// TIA Portal project "CmDrvSerPosRev0.0.5" (V15.1)

(* hardware
DEVICE "S7-1200 station_1"  S7-1200 Station
   slot 0: "Rack_0"  S7-1200 Rack  Rack  V1.0
   slot 1: "CPU"  CPU 1215C DC/DC/DC  6ES7 215-1AG40-0XB0  V4.2
DEVICE "GSD-Geraet_6"  GSD.Device.PN
   slot 0: "Baugruppenträger"  Rail  V1.0
   slot 0: "rlp_drv_ser_nip_rev1_id180303002"  E84AYCER  V 2.1
DEVICE "HMI"  TP700 Comfort
   slot 0: "HMI"  TP700 Comfort  6AV2 124-0GC01-0AX0  15.1.0.0
   slot 1: "HMI_RT_1"  TP700 Comfort  6AV2 124-0GC01-0AX0  15.1.0.0
   slot 5: "HMI.IE_CP_1"  PROFINET Interface  15.0.1.0
      slot 1: "PROFINET Interface_1"  PROFINET Interface
         slot 1: "Port_1"  Port
         slot 2: "Port_2"  Port
   slot 7: "HMI.MPI/DP_CP_1"  MPI/DP Interface  15.0.1.0
*)

// ===== PLC "CPU"  CPU 1215C DC/DC/DC =====

VAR_GLOBAL   // PLC tag table "Default tag table"
   "di_PbStart" AT %I0.0 : Bool;
   "di_PbStop" AT %I0.1 : Bool;
   "di_PbReset" AT %I0.2 : Bool;
   "di_PbJog" AT %I0.3 : Bool;
   "di_FeedbackEmStop" AT %I0.4 : Bool;   // 1 = EmStop / 0 = EmStopOK
   "dq_EnableDrive" AT %Q0.5 : Bool;
END_VAR

TYPE "stcCmDrvSerPos_CD"
   STRUCT
      iModeSet : Int;
      iStartAreaAdressErrorID : Int;   // Range between 0..64
      Commands : "stcCmCommand";
      Recipe : "stcCmDrvSerPos_RECIPE";
   END_STRUCT;
END_TYPE

TYPE "stcCmCommon_VIS"
VERSION : 0.1
   STRUCT
      stc_NewTimeToSet : Struct
         year : UInt;
         month : USInt;
         day : USInt;
         weekday : USInt;
         hour : USInt;
         minute : USInt;
         iq_bRequestLoadNewTime : Bool;
      END_STRUCT;
      q_dtlActualPlcSystemTime : DTL;
      q_rActualPlcCycleTime_Sec : Real;
   END_STRUCT;
END_TYPE

TYPE "stcCmCommon_SW"
VERSION : 0.1
   STRUCT
      q_dtlActualPlcSystem_Time : DTL;
      q_rActualPlcCycleTime_Sec : Real;
      q_bSyncBlink : Bool;   // Signal light Indicator blink
      q_bSyncBlinkText : Bool;   // Hmi status text scroll, swap, refresh blink
      q_bSyncPulsText : Bool;   // Puls is true for one cpu cycle
      q_bAlwaysTrue : Bool := TRUE;
      q_bAlwaysFalse : Bool := FALSE;
   END_STRUCT;
END_TYPE

TYPE "stcCmDrvSerPos_VIS"
   STRUCT
      Commands : "stcCmCommand";
      Interlocks : "stcCmCommand";
      Indicators : "stcCmIndicators";
      Recipe : "stcCmDrvSerPos_RECIPE";
      Settings : "stcCmDrvSerPos_CFG";
      CD : "stcCmDrvSerPos_CD";
      SD : "stcCmDrvSerPos_SD";
      bLimitsSwitchPositiveActivated : Bool;   // Module specific
      bLimitsSwitchNegativeActivated : Bool;   // Module specific
      bHomingSensorActivated : Bool;   // Module specific
   END_STRUCT;
END_TYPE

TYPE "stcCmDrvSerPos_RETAIN"
   STRUCT
      Recipe : "stcCmDrvSerPos_RECIPE";
      Settings : "stcCmDrvSerPos_CFG";
      ErrorWarningReleased : Bool;
   END_STRUCT;
END_TYPE

TYPE "stcCmDrvSerPos_RECIPE"
   STRUCT
      rSpPosition_Units : Real;
   END_STRUCT;
END_TYPE

TYPE "stcCmDrvSerPos_CFG"
   STRUCT
      rSpLimitH_Units : Real;
      rSpLimitL_Units : Real;
      rSpPositionOffset_Units : Real;
      iSetUnits : Int;   // 0=um, 1=mm, 2=cm, 10=mil, 11=Inch, 12=foot
   END_STRUCT;
END_TYPE

TYPE "stcCmDrvSerPos_SD"
   STRUCT
      iModeActual : Int;
      iModuleState : Int;
      bRFR : Bool;   // Ready for run AND active mode is Automatic
      bExecuting : Bool;   // PosCtrl executing = Executing production AND , active mode is Automatic
      bRecipeAccepted : Bool;   // Recipe as setpoints are accepted and equal with active internal setpoints
      ErrorWarningReleased : Bool;   // ErrorWarning enabled
      CommandsActivated : "stcCmCommand";   // Feedback of commands while there are activated in the StateCases
      Recipe : "stcCmDrvSerPos_RECIPE";
      ProcessValue : "stcCmDrvSerPos_PROCESS";
      ErrorWarning : "stcCmErrorWarning";
   END_STRUCT;
END_TYPE

TYPE "stcCmDrvSerPos_REMOTE"
   STRUCT
      ErrorID : DInt;
      iModuleState : Int;
      Recipe : "stcCmDrvSerPos_RECIPE";
      Process : "stcCmDrvSerPos_PROCESS";
   END_STRUCT;
END_TYPE

TYPE "stcCmDrvSerPos_PROCESS"
   STRUCT
      rPvPosition_Units : Real;
   END_STRUCT;
END_TYPE

// folder: OEM

TYPE "stcLCB_12x_SetAxisData_Sw"
VERSION : 0.1
   STRUCT
      rUnitsToPos : Real;
      rPosToUnits : Real;
   END_STRUCT;
END_TYPE

// folder: Template_ControlModule

TYPE "stcCmStates"
   STRUCT
      iModule : Int;
      iInit : Int;   // Initializing/PowerUp
      iReady : Int;
      iEnableDisable : Int;
      iJogFwdCwUpLoading : Int;
      iJogRevCcwDownUnloading : Int;
      iHoming : Int;
      iExecutingAutomatic : Int;   // Position control active, Conveyor is executing, Cutter is executing
      iError : Int;
   END_STRUCT;
END_TYPE

TYPE "stcCmCommand"
   STRUCT
      ModeChange : Bool;
      Enable : Bool;
      Disable : Bool;
      JogFwdCwUpLoading : Bool;
      JogRevCcwDownUnloading : Bool;
      StartHoming : Bool;
      StopHoming : Bool;
      StartExecuteAutomatic : Bool;   // Position control active, Conveyor is executing, Cutter is executing
      StopExecuteAutomatic : Bool;   // Position control active, Conveyor is executing, Cutter is executing
      EnableReleaseErrorWarning : Bool;
      DisableReleaseErrorWarning : Bool;
      ExecuteLoadRecipe : Bool;   // Execute module to recipe value
      ManualToAutomatic : Bool;   // Set module from Temporarily Manual control into automatic so it is reacting at commands from heigher layer
      AutomaticToManual : Bool;   // Temporarily Set module from Automatic into Manual control. The module react at VIS commands and not from heigher layer commands
      PbReset : Bool;
      PbSingleStep : Bool;   // At falling edge of the push button, the single step command will react in mode=5=SingleStepMode
   END_STRUCT;
END_TYPE

TYPE "stcCmIndicators"
   STRUCT
      PushButtons : "stcCmCommand";
      Status : Struct
         IsEnabled : Bool;
         IsHomed : Bool;
         BusyJogFwdCwUpLoading : Bool;
         BusyJogRevCcwDownUnloading : Bool;
         IsAtTargetPosSpeed : Bool;
      END_STRUCT;
   END_STRUCT;
END_TYPE

TYPE "stcCmErrorWarning"
   STRUCT
      diModuleErrorID : DInt;   // bit0-15=ErrorID, bit16-25ErrorSubjectArea, bit26-31 location area
      bErrorTripped : Bool;   // There is one or more error's going on
      bWarningTripped : Bool;   // There is one or more warning's going on
      wError : Word;   // 16 bit word. Each idividual bit stands for a item
      wWarning : Word;   // 16 bit word. Each idividual bit stands for a item
      iAdressAreaSize : Int;   // Range 0..64. the count of error location areas inside the module
   END_STRUCT;
END_TYPE

// folder: (top level)

DATA_BLOCK "DB_CmCommon"   // DB1
{ S7_Optimized_Access := 'TRUE' }
VERSION : 0.1
// stored: InstanceOfName CmCommon
"CmCommon"
BEGIN
END_DATA_BLOCK

DATA_BLOCK "DB_CmDrvSerPos"   // DB2
{ S7_Optimized_Access := 'TRUE' }
VERSION : 0.1
// stored: InstanceOfName CmDrvSerPos
"CmDrvSerPos"
BEGIN
END_DATA_BLOCK

DATA_BLOCK "VIS_CmDrvSerPos"   // DB3
{ S7_Optimized_Access := 'TRUE' }
VERSION : 0.1
   VAR
      stc : "stcCmDrvSerPos_VIS";
   END_VAR
BEGIN
END_DATA_BLOCK

DATA_BLOCK "VIS_CmCommon"   // DB4
{ S7_Optimized_Access := 'TRUE' }
VERSION : 0.1
   VAR
      stc : "stcCmCommon_VIS";
   END_VAR
BEGIN
END_DATA_BLOCK

DATA_BLOCK "RETAIN_CmDrvSerPos"   // DB5
{ S7_Optimized_Access := 'TRUE' }
VERSION : 0.1
   VAR RETAIN
      stc : "stcCmDrvSerPos_RETAIN";
   END_VAR
BEGIN
   stc.Recipe.rSpPosition_Units := 150.0;
   stc.Settings.rSpLimitH_Units := 300.0;
   stc.Settings.rSpLimitL_Units := 4.0;
   stc.Settings.rSpPositionOffset_Units := -1.8;
   stc.Settings.iSetUnits := 0;
END_DATA_BLOCK

FUNCTION_BLOCK "CmDrvSerPos"   // FB1, FBD
TITLE = Control Module: Drive Servo Positioning OEM: LENZE
{ S7_Optimized_Access := 'TRUE' }
VERSION : 0.1
   VAR_INPUT
      i_HW_IO_Head : Hw_Io;
      i_bPbReset : Bool;
      i_bQuickStop : Bool;   // True is quickstop situation active, False is normal operating
      i_bPbSingleStep : Bool;   // At falling edge of the push button, the single step command will react in mode=5=SingleStepMode
      i_JogFwdCwUpLoading : Bool;
      i_JogRevCcwDownUnloading : Bool;
      Common : "stcCmCommon_SW";
      CD : "stcCmDrvSerPos_CD";
   END_VAR
   VAR_OUTPUT
      SD : "stcCmDrvSerPos_SD";
      q_bDriveIEnableRfr : Bool;   // True=Drive from InhibitSleepMode into RFR, False=Inhibit Sleep situation en drive stopped functioning
   END_VAR
   VAR_IN_OUT
      VIS : "stcCmDrvSerPos_VIS";
      RETAIN : "stcCmDrvSerPos_RETAIN";
   END_VAR
   VAR
      RM : "stcCmDrvSerPos_CD";
      FM : Struct
         Interlock : "stcCmCommand";
         ModeActual : Int;
      END_STRUCT;
      FS : Struct
         StateCases : "stcCmStates";
         StateCasesPrevious : "stcCmStates";
         Commands : "stcCmCommand";
         CommandsActive : "stcCmCommand";
         Indicators : "stcCmIndicators";
         Settings : "stcCmDrvSerPos_CFG";
         Recipe : "stcCmDrvSerPos_RECIPE";
         ProcessValues : "stcCmDrvSerPos_PROCESS";
         ErrorWarningModule : "stcCmErrorWarning";
         ErrorWarning : "stcCmErrorWarning";
         Intern : Struct
            rPreviousSpPosition_Units : Real;
            ErrorWarningReleased : Bool;
            ErrorWarning : Struct
               wErrorLocationArea : Word;
               wErrorSubjectArea : Word;
               wErrorID : Word;
               dwModuleErrorID : DWord;
               bErrorTripped : Bool;
               bWarningTripped : Bool;
            END_STRUCT;
         END_STRUCT;
         Outputs : Struct
            bDriveInhibitTerminal : Bool;   // True=Drive from InhibitSleepMode into RFR, False=Inhibit Sleep situation en drive stopped functioning
         END_STRUCT;
      END_STRUCT;
      InstanceOEM_LCB_12x_SetAxisData : "LCB_12x_SetAxisData";
      InstanceOEM_LCB_12x_TablePositioning_V2 : "LCB_12x_TablePositioning_V2";
      InstanceF_TRIG_PbSingleStep : F_TRIG;
      InstanceR_TRIG_cmdEnable : R_TRIG;
      InstanceR_TRIG_cmdDisable : R_TRIG;
      InstanceR_TRIG_cmdStartHoming : R_TRIG;
      InstanceR_TRIG_cmdStopHoming : R_TRIG;
      InstanceR_TRIG_cmdStartExecAutomatic : R_TRIG;
      InstanceR_TRIG_cmdStopExecAutomatic : R_TRIG;
      InstanceR_TRIG_cmdLoadRecipe : R_TRIG;
   END_VAR
BEGIN

REGION Network 1 (SCL): Resource Manager
   // Mapping data channels --> Data channel switch depending of actual Mode
   CASE #FM.ModeActual OF

       0: //Wrong Mode
           #RM.iModeSet := #CD.iModeSet;
           //
           #RM.Commands.ModeChange := #CD.Commands.ModeChange;
           #RM.Commands.Enable :=
           #RM.Commands.Disable :=
           #RM.Commands.JogFwdCwUpLoading :=
           #RM.Commands.JogRevCcwDownUnloading :=
           #RM.Commands.StartHoming :=
           #RM.Commands.StopHoming :=
           #RM.Commands.StartExecuteAutomatic :=
           #RM.Commands.StopExecuteAutomatic :=
           #RM.Commands.EnableReleaseErrorWarning :=
           #RM.Commands.DisableReleaseErrorWarning :=
           #RM.Commands.ExecuteLoadRecipe :=
           #RM.Commands.ManualToAutomatic :=
           #RM.Commands.AutomaticToManual := FALSE;
           #RM.Commands.PbReset :=
               #CD.Commands.PbReset OR
               #VIS.Commands.PbReset OR
               #i_bPbReset;
           #RM.Commands.PbSingleStep := FALSE;

       1: //Automatic Inline
           #RM.iModeSet := #CD.iModeSet;
           #RM.Commands := #CD.Commands;
           //Overrule single commands
           #RM.Commands.PbReset :=
               #CD.Commands.PbReset OR
               #VIS.Commands.PbReset OR
               #i_bPbReset;

       2: //Automatic standalone
           #RM.iModeSet := #CD.iModeSet;
           #RM.Commands := #CD.Commands;
           //Overrule single commands
           #RM.Commands.PbReset :=
               #CD.Commands.PbReset OR
               #VIS.Commands.PbReset OR
               #i_bPbReset;

       3: //Manual
           #RM.iModeSet := #CD.iModeSet;
           #RM.Commands := #VIS.Commands;
           #RM.Commands.ModeChange := #CD.Commands.ModeChange;
           //Overrule single commands
           #RM.Commands.PbReset :=
               #CD.Commands.PbReset OR
               #VIS.Commands.PbReset OR
               #i_bPbReset;
           #RM.Commands.JogFwdCwUpLoading :=
               #VIS.Commands.JogFwdCwUpLoading OR
               #CD.Commands.JogFwdCwUpLoading OR
               #i_JogFwdCwUpLoading;
           #RM.Commands.JogRevCcwDownUnloading :=
               #VIS.Commands.JogRevCcwDownUnloading OR
               #CD.Commands.JogRevCcwDownUnloading OR
               #i_JogRevCcwDownUnloading;

       4: //Service
           #RM.iModeSet := #CD.iModeSet;
           #RM.Commands := #VIS.Commands;
           #RM.Commands.ModeChange := #CD.Commands.ModeChange;
           //Overrule single commands
           #RM.Commands.PbReset :=
               #CD.Commands.PbReset OR
               #VIS.Commands.PbReset OR
               #i_bPbReset;
           #RM.Commands.JogFwdCwUpLoading :=
               #VIS.Commands.JogFwdCwUpLoading OR
               #CD.Commands.JogFwdCwUpLoading OR
               #i_JogFwdCwUpLoading;
           #RM.Commands.JogRevCcwDownUnloading :=
               #VIS.Commands.JogRevCcwDownUnloading OR
               #CD.Commands.JogRevCcwDownUnloading OR
               #i_JogRevCcwDownUnloading;

       5: //SingleStep
           #RM.iModeSet := #CD.iModeSet;
           #RM.Commands := #VIS.Commands;
           #RM.Commands.ModeChange := #CD.Commands.ModeChange;
           //Overrule single commands
           #RM.Commands.PbReset :=
               #CD.Commands.PbReset OR
               #VIS.Commands.PbReset OR
               #i_bPbReset;
           #RM.Commands.JogFwdCwUpLoading :=
               #VIS.Commands.JogFwdCwUpLoading OR
               #CD.Commands.JogFwdCwUpLoading OR
               #i_JogFwdCwUpLoading;
           #RM.Commands.JogRevCcwDownUnloading :=
               #VIS.Commands.JogRevCcwDownUnloading OR
               #CD.Commands.JogRevCcwDownUnloading OR
               #i_JogRevCcwDownUnloading;
           #RM.Commands.PbReset :=
               #CD.Commands.PbReset OR
               #VIS.Commands.PbReset OR
               #i_bPbReset;
           #RM.Commands.PbSingleStep :=
               #CD.Commands.PbSingleStep OR
               #VIS.Commands.PbSingleStep OR
               #i_bPbSingleStep;
   END_CASE;
END_REGION

REGION Network 2 (SCL): Funtional Manager: Interlocks
   REGION #FM.Interlock.ModeChange
       #FM.Interlock.ModeChange :=
           (
           #FS.StateCases.iModule = 10 (*Disabled*)OR
           #FS.StateCases.iModule = 30 (*ReadyEnabled*) OR
           #FS.StateCases.iModule = 70 (*ReadyHomed*) OR
           #FS.StateCases.iModule = 80 (*Executing*) 
           );
   END_REGION

   REGION #FM.Interlock.Enable Disable
       #FM.Interlock.Disable :=
           (
           #FS.StateCases.iInit = 100 AND
           #FS.StateCases.iReady > 0 AND
           #FS.StateCases.iEnableDisable > 0 AND
           #FS.StateCases.iJogFwdCwUpLoading = 0 AND
           #FS.StateCases.iJogRevCcwDownUnloading = 0 AND
           (#FS.StateCases.iHoming = 0 OR #FS.StateCases.iHoming = 100) AND
           #FS.StateCases.iExecutingAutomatic = 0
           );

       #FM.Interlock.Enable :=
           (
           #FS.StateCases.iInit = 100 AND
           #FS.StateCases.iReady > 0 AND
           #FS.StateCases.iEnableDisable = 0 AND
           #FS.StateCases.iJogFwdCwUpLoading = 0 AND
           #FS.StateCases.iJogRevCcwDownUnloading = 0 AND
           (#FS.StateCases.iHoming = 0 OR #FS.StateCases.iHoming = 100) AND
           #FS.StateCases.iExecutingAutomatic = 0
           );
   END_REGION

   REGION #FM.Interlock.Jog
       #FM.Interlock.JogFwdCwUpLoading :=
       (
       #FM.ModeActual <> 5 (*Single step mode*)AND
       #FS.StateCases.iInit = 100 AND
       #FS.StateCases.iReady >= 20 AND
       #FS.StateCases.iEnableDisable = 100(*Executed*)AND
       // #FS.State.iJogFwdCwUp = 0 AND
       #FS.StateCases.iJogRevCcwDownUnloading = 0 AND
       (#FS.StateCases.iHoming = 0 OR #FS.StateCases.iHoming = 100 (*Executed*)) AND
       #FS.StateCases.iExecutingAutomatic = 0 AND
       (#FS.StateCases.iError = 0 (*No Error*) OR #FS.StateCases.iError >= 500) (*Warning*) AND
       NOT #InstanceOEM_LCB_12x_TablePositioning_V2.xHW_LimitSwitchPos
       );

       #FM.Interlock.JogRevCcwDownUnloading :=
       (
       #FM.ModeActual <> 5 (*Single step mode*)AND
       #FS.StateCases.iInit = 100 AND
       #FS.StateCases.iReady >= 20 AND
       #FS.StateCases.iEnableDisable = 100(*Executed*)AND
       #FS.StateCases.iJogFwdCwUpLoading = 0 AND
       //#FS.State.iJogRevCcwDown = 0 AND
       (#FS.StateCases.iHoming = 0 OR #FS.StateCases.iHoming = 100 (*Executed*)) AND
       #FS.StateCases.iExecutingAutomatic = 0 AND
       (#FS.StateCases.iError = 0 (*No Error*) OR #FS.StateCases.iError >= 500) (*Warning*) AND
       NOT #InstanceOEM_LCB_12x_TablePositioning_V2.xHW_LimitSwitchNeg
       );
   END_REGION

   REGION #FM.Interlock.Homing Start Stop
       #FM.Interlock.StartHoming :=
           (
           #FS.StateCases.iInit = 100 AND
           #FS.StateCases.iReady >= 20 AND
           #FS.StateCases.iEnableDisable = 100(*Executed*)AND
           #FS.StateCases.iJogFwdCwUpLoading = 0 AND
           #FS.StateCases.iJogRevCcwDownUnloading = 0 AND
           (#FS.StateCases.iHoming = 0 OR #FS.StateCases.iHoming = 100 (*Executed*)) AND
           #FS.StateCases.iExecutingAutomatic = 0 AND
           #FS.StateCases.iError = 0
           );

       #FM.Interlock.StopHoming :=
           (
           #FS.StateCases.iInit = 100 AND
           #FS.StateCases.iReady >= 20 AND
           #FS.StateCases.iEnableDisable = 100(*Executed*)AND
           #FS.StateCases.iJogFwdCwUpLoading = 0 AND
           #FS.StateCases.iJogRevCcwDownUnloading = 0 AND
           #FS.StateCases.iHoming > 0 (*Stopped*) AND
           #FS.StateCases.iExecutingAutomatic = 0 AND
           #FS.StateCases.iError = 0
           );
   END_REGION

   REGION #FM.Interlock.PositionControl Start Stop
       #FM.Interlock.StartExecuteAutomatic :=
           (
           #FS.StateCases.iInit = 100 AND
           #FS.StateCases.iReady >= 30 AND
           #FS.StateCases.iEnableDisable = 100(*Executed*)AND
           #FS.StateCases.iJogFwdCwUpLoading = 0 AND
           #FS.StateCases.iJogRevCcwDownUnloading = 0 AND
           #FS.StateCases.iHoming = 100 (*Executed*) AND
           #FS.StateCases.iExecutingAutomatic = 0 (*Stopped*)AND
           #FS.StateCases.iError = 0
           );

       #FM.Interlock.StopExecuteAutomatic :=
           (
           #FS.StateCases.iInit = 100 AND
           //#FS.State.iReady > 0 AND
           #FS.StateCases.iEnableDisable = 100(*Executed*)AND
           #FS.StateCases.iJogFwdCwUpLoading = 0 AND
           #FS.StateCases.iJogRevCcwDownUnloading = 0 AND
           #FS.StateCases.iHoming = 100 (*Executed*)AND
           #FS.StateCases.iExecutingAutomatic > 0 (*Stopped*) AND
           #FS.StateCases.iError = 0
           );
   END_REGION

   REGION #FM.Interlock.ReleaseErrorWarning
       #FM.Interlock.EnableReleaseErrorWarning :=
           (
           #FS.StateCases.iInit = 100
           );

       #FM.Interlock.DisableReleaseErrorWarning :=
           (
           #FS.StateCases.iInit = 100
           );
   END_REGION

   REGION #FM.Interlock.LoadRecipe
       #FM.Interlock.ExecuteLoadRecipe :=
           (
           #FM.ModeActual = 1 OR
           #FM.ModeActual = 2 OR
           #FM.ModeActual = 3 OR
           #FM.ModeActual = 4 OR
           #FM.ModeActual = 5
           );
   END_REGION

   REGION  #FM.Interlock.ManualToAutomatic / AutomaticToManual
       #FM.Interlock.ManualToAutomatic :=
           (
           #FS.StateCases.iReady > 0
           );

       #FM.Interlock.AutomaticToManual :=
           (
           TRUE
           );
   END_REGION

   REGION #FM.Interlock.PbReset
       #FM.Interlock.PbReset := TRUE;

   END_REGION

   REGION #FM.Interlock.PbSingleStep
   #FM.Interlock.PbSingleStep :=
       #FM.ModeActual = 5;//SingleStep Mode
   END_REGION
END_REGION

REGION Network 3 (SCL): Functional Manager: Commands
   #FS.Commands.ModeChange :=
       #FM.Interlock.ModeChange AND
       #RM.Commands.ModeChange;

   #InstanceR_TRIG_cmdEnable(CLK := #RM.Commands.Enable);
   #FS.Commands.Enable :=
       #FM.Interlock.Enable AND
       #InstanceR_TRIG_cmdEnable.Q;

   #InstanceR_TRIG_cmdDisable(CLK := #RM.Commands.Disable);
   #FS.Commands.Disable :=
       #FM.Interlock.Disable AND
       #InstanceR_TRIG_cmdDisable.Q;

   #FS.Commands.JogFwdCwUpLoading :=
       #FM.Interlock.JogFwdCwUpLoading AND
       #RM.Commands.JogFwdCwUpLoading;

   #FS.Commands.JogRevCcwDownUnloading :=
       #FM.Interlock.JogRevCcwDownUnloading AND
       #RM.Commands.JogRevCcwDownUnloading;

   #InstanceR_TRIG_cmdStartHoming(CLK := #RM.Commands.StartHoming);
   #FS.Commands.StartHoming :=
       #FM.Interlock.StartHoming AND
       #InstanceR_TRIG_cmdStartHoming.Q;

   #InstanceR_TRIG_cmdStopHoming(CLK := #RM.Commands.StopHoming);
   #FS.Commands.StopHoming :=
       #FM.Interlock.StopHoming AND
       #InstanceR_TRIG_cmdStopHoming.Q;

   #InstanceR_TRIG_cmdStartExecAutomatic(CLK := #RM.Commands.StartExecuteAutomatic);
   #FS.Commands.StartExecuteAutomatic :=
       #FM.Interlock.StartExecuteAutomatic AND 
       #InstanceR_TRIG_cmdStartExecAutomatic.Q;

   #InstanceR_TRIG_cmdStopExecAutomatic(CLK := #RM.Commands.StopExecuteAutomatic);
   #FS.Commands.StopExecuteAutomatic :=
       #FM.Interlock.StopExecuteAutomatic AND
       #InstanceR_TRIG_cmdStopExecAutomatic.Q;

   #FS.Commands.EnableReleaseErrorWarning :=
       #FM.Interlock.EnableReleaseErrorWarning AND
       #RM.Commands.EnableReleaseErrorWarning;

   #FS.Commands.DisableReleaseErrorWarning :=
       #FM.Interlock.DisableReleaseErrorWarning AND
       #RM.Commands.DisableReleaseErrorWarning;

   //#InstanceR_TRIG_cmdLoadRecipe(CLK := #RM.Commands.ExecuteLoadRecipe);
   #FS.Commands.ExecuteLoadRecipe :=
       #FM.Interlock.ExecuteLoadRecipe AND
       #RM.Commands.ExecuteLoadRecipe; //#InstanceR_TRIG_cmdLoadRecipe.Q;

   #FS.Commands.ManualToAutomatic :=
       #FM.Interlock.ManualToAutomatic AND
       #RM.Commands.ManualToAutomatic;

   #FS.Commands.AutomaticToManual :=
       #FM.Interlock.AutomaticToManual AND
       #RM.Commands.AutomaticToManual;

   #FS.Commands.PbReset :=
       #FM.Interlock.PbReset AND 
       (
       #RM.Commands.PbReset OR
       #VIS.Commands.PbReset OR
       #i_bPbReset
       );

   #InstanceF_TRIG_PbSingleStep(CLK:=#RM.Commands.PbSingleStep);
   #FS.Commands.PbSingleStep :=
       #FM.Interlock.PbSingleStep AND
       #InstanceF_TRIG_PbSingleStep.Q;
END_REGION

REGION Network 4 (SCL): Functional Manager: Recipe
   CASE #FM.ModeActual OF
       1,2,5 :
           #VIS.Recipe := #FS.Recipe := #CD.Recipe;
       3,4 :
           #FS.Recipe:= #VIS.Recipe;
       ELSE
           #FS.Recipe := #VIS.Recipe;
   END_CASE;
END_REGION

REGION Network 5 (SCL): Functional Manager: Settings Module
   #FS.Settings := #VIS.Settings;
END_REGION

REGION Network 6 (SCL): Functional Manager: Conditioning Recipe Setpoint
   REGION  Sp Limit handling   
       IF #FS.Recipe.rSpPosition_Units > #FS.Settings.rSpLimitH_Units THEN
           #FS.Recipe.rSpPosition_Units := #FS.Settings.rSpLimitH_Units;
       ELSIF #FS.Recipe.rSpPosition_Units < #FS.Settings.rSpLimitL_Units THEN
           #FS.Recipe.rSpPosition_Units := #FS.Settings.rSpLimitL_Units;
       END_IF;
   END_REGION

   REGION Calculate position control value FOR the drive
       //Calculate position control value for the drive
       //      Drive Homing position is 0mm, Down is negative Cv position for the drive,
       //      If Nip fysical=0mm then for example -300mm is drive CV value.
       #InstanceOEM_LCB_12x_TablePositioning_V2.rPositionSet :=
       #FS.Recipe.rSpPosition_Units - #FS.Settings.rSpLimitH_Units + #FS.Settings.rSpPositionOffset_Units;
   END_REGION
END_REGION

REGION Network 7 (SCL): Functional Manager: Module mode
   //Range iModeSet
   IF #RM.iModeSet < 0 THEN
       #RM.iModeSet := 0; //Wrong Mode
   ELSIF #RM.iModeSet > 5 THEN
       #RM.iModeSet := 0; //Wrong Mode
   END_IF;

   IF #FM.Interlock.ModeChange AND #FS.Commands.ModeChange THEN
       #FS.CommandsActive.ModeChange := #FS.Commands.ModeChange;
       #FM.ModeActual := #RM.iModeSet;
   ELSE
       #FS.CommandsActive.ModeChange := FALSE;
   END_IF;
END_REGION

REGION Network 8 (SCL): Functional Strategy: State Initializing / Write Retain
   CASE #FS.StateCases.iInit OF

       0: //Stopped
           //Output
           #VIS.Recipe := #FS.Recipe := #RETAIN.Recipe; //#CD.Recipe is input can not be written
           #VIS.Settings := #FS.Settings := #RETAIN.Settings;
           #FS.Intern.ErrorWarningReleased := #RETAIN.ErrorWarningReleased;
           //Transistion
           #FS.StateCases.iInit := 100;

       100: //Executed
           //Output
           #RETAIN.Recipe := #FS.Recipe;
           #RETAIN.Settings := #FS.Settings;
           #RETAIN.ErrorWarningReleased := #FS.Intern.ErrorWarningReleased;
           //Transistion

   END_CASE;
END_REGION

REGION Network 9 (SCL): Functional Strategy: SingleStep Mode--> Store Previous StateCases
   #FS.StateCasesPrevious := #FS.StateCases;
END_REGION

REGION Network 10 (SCL): Functional Strategy: State Module
   //Global Transistions handling
   IF #FS.ErrorWarning.wError <> 0 THEN
       #FS.StateCases.iModule := 90; //Error
   END_IF;

   CASE #FS.StateCases.iModule OF

       0: (* Inititialzed *)
           //Transistion
           IF #FS.StateCases.iInit = 100 THEN
               #FS.StateCases.iModule := 10; //Disabled
           END_IF;

       10: //Disabled
           //Transistion
           IF #FS.StateCases.iEnableDisable > 0 THEN
               #FS.StateCases.iModule := 20; //Enabling
           END_IF;

       20: // Enabling
           //Transistion
           IF #FS.StateCases.iEnableDisable >= 100 AND #FS.StateCases.iEnableDisable < 150 THEN //Executed
               #FS.StateCases.iModule := 30; //ReadyEnabled
           ELSIF #FS.StateCases.iEnableDisable >= 150 THEN //Stopping=Disabling
               #FS.StateCases.iModule := 25; //Disabling
           END_IF;

       25: // Disabling
           //Transistion
           IF #FS.StateCases.iEnableDisable = 0 THEN //Stopped = Disabled
               #FS.StateCases.iModule := 10; //Disabled
           ELSIF #FS.StateCases.iEnableDisable > 0 AND #FS.StateCases.iEnableDisable < 150 THEN //Busy Enabling Or is Enabled
               #FS.StateCases.iModule := 20; //Enabling
           END_IF;

       30: //ReadyEnabled
           //Transistion
           IF #FS.StateCases.iJogFwdCwUpLoading > 0 THEN
               #FS.StateCases.iModule := 40; //Jog Forward
           ELSIF #FS.StateCases.iJogRevCcwDownUnloading > 0 THEN
               #FS.StateCases.iModule := 50; //Jog Reverse
           ELSIF #FS.StateCases.iHoming > 0 THEN
               #FS.StateCases.iModule := 60; //Homing
           ELSIF #FS.StateCases.iEnableDisable >= 150 OR #FS.StateCases.iEnableDisable = 0 THEN
               #FS.StateCases.iModule := 25; //Disabling
           END_IF;

       40: //Jog Forward
           //Actions
           //Transistion
           IF #FS.StateCases.iJogFwdCwUpLoading = 0 THEN
               IF #FS.StateCases.iReady = 20 THEN //ReadyEnabled
                   #FS.StateCases.iModule := 30; //Jog Forward
               ELSIF #FS.StateCases.iReady = 30 THEN //ReadyHomed
                   #FS.StateCases.iModule := 70; //ReadyHomed
               END_IF;
           END_IF;

       50: //Jog Reverse
           //Transistions
           IF #FS.StateCases.iJogRevCcwDownUnloading = 0 THEN
               IF #FS.StateCases.iReady = 20 THEN //ReadyEnabled
                   #FS.StateCases.iModule := 30; //Jog Forward
               ELSIF #FS.StateCases.iReady = 30 THEN //ReadyHomed
                   #FS.StateCases.iModule := 70; //ReadyHomed
               END_IF;
           END_IF;

       60: //HomingBusy
           //Transistion
           IF #FS.StateCases.iHoming >= 100 AND #FS.StateCases.iHoming < 150  THEN //Is Homed
               #FS.StateCases.iModule := 70; //ReadyHomed
           ELSIF #FS.StateCases.iHoming >= 150 THEN //HomingStopping
               #FS.StateCases.iModule := 65; //HomingStopping
           END_IF;

       65: //HomingStopping
           //Transistion
           IF #FS.StateCases.iHoming = 0 THEN //Stopped
               #FS.StateCases.iModule := 30; //ReadyEnabled
           ELSIF #FS.StateCases.iHoming > 0 AND #FS.StateCases.iHoming <= 100  THEN //HomingStarting
               #FS.StateCases.iModule := 60; //ReadyHomed
           END_IF;

       70: //ReadyHomed
           //Transistion
           IF #FS.StateCases.iJogFwdCwUpLoading > 0 THEN
               #FS.StateCases.iModule := 40; //Jog Forward
           ELSIF #FS.StateCases.iJogRevCcwDownUnloading > 0 THEN
               #FS.StateCases.iModule := 50; //Jog Reverse
           ELSIF #FS.StateCases.iHoming >= 150 OR #FS.StateCases.iHoming = 0 THEN //HomingStopping
               #FS.StateCases.iModule := 65; //HomingStopping    
           ELSIF #FS.StateCases.iExecutingAutomatic > 0 THEN
               #FS.StateCases.iModule := 80; //PostionControl
           ELSIF #FS.StateCases.iEnableDisable >= 150 OR #FS.StateCases.iEnableDisable = 0 THEN
               #FS.StateCases.iModule := 25; //Disabling
           END_IF;

       80: //Executing (PositionControlBusy)
          //Transistion
           IF #FS.StateCases.iExecutingAutomatic >= 150 OR #FS.StateCases.iExecutingAutomatic = 0 THEN
               #FS.StateCases.iModule := 85; //ExecutingStopping
           END_IF;

       85: //ExecutingStopping (PostionControlStopping)
           //Transistion
           IF #FS.StateCases.iExecutingAutomatic = 0 THEN
               #FS.StateCases.iModule := 70; //ReadyHomed
           END_IF;

       90: //Error
           //Transistion
           IF #FS.ErrorWarning.wError = 0 THEN
               #FS.StateCases.iModule := 0; //Stopped
           END_IF;
   END_CASE;
END_REGION

REGION Network 11 (SCL): Functional Strategy: State Ready
   CASE #FS.StateCases.iReady OF

       0: //Disabled
           //Transistion
           IF  #FS.StateCases.iInit = 100 AND
               #FS.StateCases.iEnableDisable = 0
           THEN
               #FS.StateCases.iReady := 10; //Ready from disabled, wait for Enable
           END_IF;

       10: //ReadyDisabled, wait for Enable
           //Transistions
           IF #FS.StateCases.iEnableDisable = 100(*Executed*)THEN
               #FS.StateCases.iReady := 20; //Ready and Is Enabled, wait for Homing
           ELSIF #FS.StateCases.iInit <> 100 THEN
               #FS.StateCases.iReady := 0; //Disabled
           END_IF;

       20: //ReadyEnabled, wait for Homing
           //Transistion
           IF #FS.StateCases.iInit = 100(*Executed*) AND
               #FS.StateCases.iEnableDisable = 100(*Executed*)AND
               #FS.StateCases.iHoming = 100 (*Executed*)
           THEN
               #FS.StateCases.iReady := 30;
           ELSIF #FS.StateCases.iInit <> 100(*Executed*) OR
               #FS.StateCases.iEnableDisable <> 100(*Executed*)
           THEN
               #FS.StateCases.iReady := 10;
           END_IF;

       30: //Ready and Is Homed, ready for position control
           //Transistion
           IF  #FS.StateCases.iInit <> 100(*Executed*) OR
               #FS.StateCases.iEnableDisable <> 100(*Executed*)OR
               #FS.StateCases.iHoming <> 100 (*Executed*)
           THEN
               #FS.StateCases.iReady := 20;
           END_IF;
   END_CASE;
END_REGION

REGION Network 12 (SCL): Functional Strategy: State EnableDisable
   CASE #FS.StateCases.iEnableDisable OF

       0: //Stopped
           //Actions
           #FS.CommandsActive.Enable := FALSE;
           #FS.CommandsActive.Disable := FALSE;
           //
           #FS.Indicators.PushButtons.Enable := FALSE;
           #FS.Indicators.PushButtons.Disable := FALSE;
           #FS.Indicators.Status.IsEnabled := FALSE;
           //
           #InstanceOEM_LCB_12x_TablePositioning_V2.xDriveEnable := FALSE;
           //Transistion
           IF #FS.Commands.Enable AND NOT #FS.Commands.Disable THEN //Disable higher prio then Enable
               #FS.StateCases.iEnableDisable := 10; //Starting, Get Drive from inhibit(Sleep) state
           END_IF;

       10: //Starting, Get Drive from inhibit(Sleep) state
           //Actions
           #FS.CommandsActive.Enable := #FS.Commands.Enable;
           #FS.CommandsActive.Disable := FALSE;
           //
           #FS.Indicators.PushButtons.Enable := TRUE;
           #FS.Indicators.PushButtons.Disable := FALSE;
           #FS.Indicators.Status.IsEnabled := FALSE;
           //
           #FS.Outputs.bDriveInhibitTerminal := TRUE;
           #InstanceOEM_LCB_12x_TablePositioning_V2.xDriveEnable := FALSE;
           //Transistion
           IF #InstanceOEM_LCB_12x_TablePositioning_V2.xDriveReady THEN
               #FS.StateCases.iEnableDisable := 11; //Starting, Enabling
           ELSIF #FS.Commands.Disable THEN
               #FS.StateCases.iEnableDisable := 150; //Stopping
           END_IF;

       11: //Starting, Enabling
           //Actions
           #FS.CommandsActive.Enable := #FS.Commands.Enable;
           #FS.CommandsActive.Disable := FALSE;
           //
           #FS.Indicators.PushButtons.Enable := TRUE;
           #FS.Indicators.PushButtons.Disable := FALSE;
           #FS.Indicators.Status.IsEnabled := FALSE;
           //
           #FS.Outputs.bDriveInhibitTerminal := TRUE;
           #InstanceOEM_LCB_12x_TablePositioning_V2.xDriveEnable := TRUE;
           //Transistion
           IF #InstanceOEM_LCB_12x_TablePositioning_V2.xDriveEnabled THEN
               #FS.StateCases.iEnableDisable := 50; //Executing
           ELSIF #FS.Commands.Disable THEN
               #FS.StateCases.iEnableDisable := 150; //Stopping
           END_IF;

       50: //Executing
           //Actions
           #FS.CommandsActive.Enable := #FS.Commands.Enable;
           #FS.CommandsActive.Disable := FALSE;
           //
           #FS.Indicators.PushButtons.Enable := TRUE;
           #FS.Indicators.PushButtons.Disable := FALSE;
           #FS.Indicators.Status.IsEnabled := FALSE;
           //
           #InstanceOEM_LCB_12x_TablePositioning_V2.xDriveEnable := TRUE;
           //Transistion
           IF #InstanceOEM_LCB_12x_TablePositioning_V2.xDriveEnabled THEN
               #FS.StateCases.iEnableDisable := 100; //Ready and Is Enabled, wait for Homing
           ELSIF #FS.Commands.Disable THEN
               #FS.StateCases.iEnableDisable := 150; //Stopping
           END_IF;

       100://Executed
           //Actions
           #FS.CommandsActive.Enable := #FS.Commands.Enable;
           #FS.CommandsActive.Disable := FALSE;
           //
           #FS.Indicators.PushButtons.Enable := #FS.CommandsActive.Enable;
           #FS.Indicators.PushButtons.Disable := FALSE;
           #FS.Indicators.Status.IsEnabled := TRUE;
           //
           //Transistion
           IF #FS.Commands.Disable THEN //Disable higher prio then Enable
               #FS.StateCases.iEnableDisable := 150; //Stopping
           END_IF;

       150: //Stopping
           //Actions
           #FS.CommandsActive.Enable := FALSE;
           #FS.CommandsActive.Disable := #FS.Commands.Disable;
           //
           #FS.Indicators.PushButtons.Enable := FALSE;
           #FS.Indicators.PushButtons.Disable := TRUE;
           #FS.Indicators.Status.IsEnabled := FALSE;
           //
           #FS.Outputs.bDriveInhibitTerminal := TRUE;
           #InstanceOEM_LCB_12x_TablePositioning_V2.xDriveEnable := FALSE;
           //Transistion
           IF NOT #InstanceOEM_LCB_12x_TablePositioning_V2.xDriveEnabled THEN
               #FS.StateCases.iEnableDisable := 151; //Stopping, Set drive inhibit(sleep) mode
           END_IF;

       151: //Stopping, Set drive inhibit(sleep) mode
           //Actions
           #FS.CommandsActive.Enable := FALSE;
           #FS.CommandsActive.Disable := #FS.Commands.Disable;
           //
           #FS.Indicators.PushButtons.Enable := FALSE;
           #FS.Indicators.PushButtons.Disable := TRUE;
           #FS.Indicators.Status.IsEnabled := FALSE;
           //
           #FS.Outputs.bDriveInhibitTerminal := FALSE;
           #InstanceOEM_LCB_12x_TablePositioning_V2.xDriveEnable := FALSE;
           //Transistion
           IF NOT #InstanceOEM_LCB_12x_TablePositioning_V2.xDriveEnabled THEN
               #FS.StateCases.iEnableDisable := 0; //Inititialzed
           END_IF;
   END_CASE;
END_REGION

REGION Network 13 (SCL): Functional Strategy: State JogFwdCwUpLoading
   CASE #FS.StateCases.iJogFwdCwUpLoading OF

       0: //Stopped
           //Actions
           #FS.CommandsActive.JogFwdCwUpLoading := FALSE;
           //
           #FS.Indicators.PushButtons.JogFwdCwUpLoading := FALSE;
           #FS.Indicators.Status.BusyJogFwdCwUpLoading := FALSE;
           //
           #InstanceOEM_LCB_12x_TablePositioning_V2.xManualPos := False;
           //Transistion
           IF #FS.Commands.JogFwdCwUpLoading THEN
               #FS.StateCases.iJogFwdCwUpLoading := 10;
           END_IF;

       10: //Starting
           //Actions
           #FS.CommandsActive.JogFwdCwUpLoading := #FS.Commands.JogFwdCwUpLoading;
           //
           #FS.Indicators.PushButtons.JogFwdCwUpLoading := TRUE;
           #FS.Indicators.Status.BusyJogFwdCwUpLoading := TRUE;
           //
           #InstanceOEM_LCB_12x_TablePositioning_V2.xManualPos := TRUE;
           //Transistion
           IF NOT #FS.Commands.JogFwdCwUpLoading THEN
               #FS.StateCases.iJogFwdCwUpLoading := 150; //Stopping
           ELSIF NOT #InstanceOEM_LCB_12x_TablePositioning_V2.xSpeedEqZero THEN
               #FS.StateCases.iJogFwdCwUpLoading := 50; //Executing
           END_IF;

       50://Executing
           //Actions
           #FS.CommandsActive.JogFwdCwUpLoading := #FS.Commands.JogFwdCwUpLoading;
           //
           #FS.Indicators.PushButtons.JogFwdCwUpLoading := TRUE;
           #FS.Indicators.Status.BusyJogFwdCwUpLoading := TRUE;
           //
           #InstanceOEM_LCB_12x_TablePositioning_V2.xManualPos := TRUE;
           //Transistion
           IF NOT #FS.Commands.JogFwdCwUpLoading THEN
               #FS.StateCases.iJogFwdCwUpLoading := 150; //Stopping
           ELSIF #InstanceOEM_LCB_12x_TablePositioning_V2.xSpeedEqZero THEN
               #FS.StateCases.iJogFwdCwUpLoading := 150; //Stopping
           END_IF;

       150: //Stopping        
           //Actions
           #FS.CommandsActive.JogFwdCwUpLoading := #FS.Commands.JogFwdCwUpLoading;
           //
           #FS.Indicators.PushButtons.JogFwdCwUpLoading := FALSE;
           #FS.Indicators.Status.BusyJogFwdCwUpLoading := TRUE;
           //
           #InstanceOEM_LCB_12x_TablePositioning_V2.xManualPos := FALSE;
           //Transistion
          IF #InstanceOEM_LCB_12x_TablePositioning_V2.xSpeedEqZero THEN
               #FS.StateCases.iJogFwdCwUpLoading := 0; //Stopped
          END_IF;
   END_CASE;
END_REGION

REGION Network 14 (SCL): Functional Strategy: State JogRevCcwDownUnloading
   CASE #FS.StateCases.iJogRevCcwDownUnloading OF

       0: //Stopped
           //Actions
           #FS.CommandsActive.JogRevCcwDownUnloading := FALSE;
           //
           #FS.Indicators.PushButtons.JogRevCcwDownUnloading := FALSE;
           #FS.Indicators.Status.BusyJogRevCcwDownUnloading := FALSE;
           //
           #InstanceOEM_LCB_12x_TablePositioning_V2.xManualNeg := False;
           //Transistion
           IF #FS.Commands.JogRevCcwDownUnloading THEN
               #FS.StateCases.iJogRevCcwDownUnloading := 10;
           END_IF;

       10: //Starting
           //Actions
           #FS.CommandsActive.JogRevCcwDownUnloading := #FS.Commands.JogRevCcwDownUnloading;
           //
           #FS.Indicators.PushButtons.JogRevCcwDownUnloading := TRUE;
           #FS.Indicators.Status.BusyJogRevCcwDownUnloading := TRUE;
           //
           #InstanceOEM_LCB_12x_TablePositioning_V2.xManualNeg := TRUE;
           //Transistion
           IF NOT #FS.Commands.JogRevCcwDownUnloading THEN
               #FS.StateCases.iJogRevCcwDownUnloading := 150; //Stopping
           ELSIF NOT #InstanceOEM_LCB_12x_TablePositioning_V2.xSpeedEqZero THEN
               #FS.StateCases.iJogRevCcwDownUnloading := 50; //Executing
           END_IF;

       50://Executing
           //Actions
           #FS.CommandsActive.JogRevCcwDownUnloading := #FS.Commands.JogRevCcwDownUnloading;
           //
           #FS.Indicators.PushButtons.JogRevCcwDownUnloading := TRUE;
           #FS.Indicators.Status.BusyJogRevCcwDownUnloading := TRUE;
           //
           #InstanceOEM_LCB_12x_TablePositioning_V2.xManualNeg := TRUE;
           //Transistion
           IF NOT #FS.Commands.JogRevCcwDownUnloading THEN
               #FS.StateCases.iJogRevCcwDownUnloading := 150; //Stopping
           ELSIF #InstanceOEM_LCB_12x_TablePositioning_V2.xSpeedEqZero THEN
               #FS.StateCases.iJogRevCcwDownUnloading := 150; //Executing
           END_IF;

       150: //Stopping        
           //Actions
           #FS.CommandsActive.JogRevCcwDownUnloading := #FS.Commands.JogRevCcwDownUnloading;
           //
           #FS.Indicators.PushButtons.JogRevCcwDownUnloading := FALSE;
           #FS.Indicators.Status.BusyJogRevCcwDownUnloading := TRUE;
           //
           #InstanceOEM_LCB_12x_TablePositioning_V2.xManualNeg := FALSE;
           //Transistion
          IF #InstanceOEM_LCB_12x_TablePositioning_V2.xSpeedEqZero THEN
              #FS.StateCases.iJogRevCcwDownUnloading := 0; //Stopped
          END_IF;
   END_CASE;
END_REGION

REGION Network 15 (SCL): Functional Strategy: State Homing
   CASE #FS.StateCases.iHoming OF
       0: //Stopped
           //Actions
           #FS.CommandsActive.StartHoming := FALSE;
           #FS.CommandsActive.StopHoming := FALSE;
           //
           #FS.Indicators.PushButtons.StartHoming := FALSE;
           #FS.Indicators.PushButtons.StopHoming := FALSE;
           #FS.Indicators.Status.IsHomed := FALSE;
           //
           #InstanceOEM_LCB_12x_TablePositioning_V2.xHomingReset := FALSE;
           #InstanceOEM_LCB_12x_TablePositioning_V2.xHomingStart := FALSE;

           //Transistions
           IF #FS.Commands.StartHoming THEN
               #FS.StateCases.iHoming := 10;//Starting
           END_IF;

       10: //Starting, Reset home position
           //Actions
           #FS.CommandsActive.StartHoming := #FS.Commands.StartHoming;
           #FS.CommandsActive.StopHoming := FALSE;
           //
           #FS.Indicators.PushButtons.StartHoming := TRUE;
           #FS.Indicators.PushButtons.StopHoming := FALSE;
           #FS.Indicators.Status.IsHomed := FALSE;
           //
           #InstanceOEM_LCB_12x_TablePositioning_V2.xHomingReset := TRUE;
           //Transistions
           IF NOT #InstanceOEM_LCB_12x_TablePositioning_V2.xHomingDone THEN
               #FS.StateCases.iHoming := 11;//Starting
           ELSIF #FS.Commands.StopHoming THEN
               #FS.StateCases.iHoming := 150; //Stopping            
           END_IF;

       11: // Starting, Set Homing profile number
           //Actions
           #FS.CommandsActive.StartHoming := #FS.Commands.StartHoming;
           #FS.CommandsActive.StopHoming := FALSE;
           //
           #FS.Indicators.PushButtons.StartHoming := TRUE;
           #FS.Indicators.PushButtons.StopHoming := FALSE;
           #FS.Indicators.Status.IsHomed := FALSE;
           //
           #InstanceOEM_LCB_12x_TablePositioning_V2.xHomingReset := FALSE;
           #InstanceOEM_LCB_12x_TablePositioning_V2.wProfileNumberSet := 1;
           //Transistions
           #FS.StateCases.iHoming := 12;//Starting

       12: //Starting, Start homing motion
           //Actions
           #FS.CommandsActive.StartHoming := #FS.Commands.StartHoming;
           #FS.CommandsActive.StopHoming := FALSE;
           //
           #FS.Indicators.PushButtons.StartHoming := TRUE;
           #FS.Indicators.PushButtons.StopHoming := FALSE;
           #FS.Indicators.Status.IsHomed := FALSE;
           //
           #InstanceOEM_LCB_12x_TablePositioning_V2.wProfileNumberSet := 1;
           #InstanceOEM_LCB_12x_TablePositioning_V2.xHomingStart := TRUE;
           //Transistions
           IF #InstanceOEM_LCB_12x_TablePositioning_V2.xHomingActive THEN
               #FS.StateCases.iHoming := 50;//Executing
           ELSIF #FS.Commands.StopHoming THEN
               #FS.StateCases.iHoming := 150; //Stopping            
           END_IF;

       50: //Executing, Wait limit switch is reached
           //Actions
           #FS.CommandsActive.StartHoming := #FS.Commands.StartHoming;
           #FS.CommandsActive.StopHoming := FALSE;
           //
           #FS.Indicators.PushButtons.StartHoming := TRUE;
           #FS.Indicators.PushButtons.StopHoming := FALSE;
           #FS.Indicators.Status.IsHomed := FALSE;
           //
           #InstanceOEM_LCB_12x_TablePositioning_V2.wProfileNumberSet := 1;
           #InstanceOEM_LCB_12x_TablePositioning_V2.xHomingStart := TRUE;
           //Transistions
           IF #InstanceOEM_LCB_12x_TablePositioning_V2.xHomingDone THEN
               #FS.StateCases.iHoming := 52;//Executed    
           ELSIF #InstanceOEM_LCB_12x_TablePositioning_V2.xDirectionSpeedIsCcw THEN
               #FS.StateCases.iHoming := 51;//Executing
           ELSIF #FS.Commands.StopHoming THEN
               #FS.StateCases.iHoming := 150; //Stopping            
           END_IF;

       51: //Executing, Wait at falling edge homing sensor        
           //Actions
           #FS.CommandsActive.StartHoming := #FS.Commands.StartHoming;
           #FS.CommandsActive.StopHoming := FALSE;
           //
           #FS.Indicators.PushButtons.StartHoming := TRUE;
           #FS.Indicators.PushButtons.StopHoming := FALSE;
           #FS.Indicators.Status.IsHomed := FALSE;
           //
           #InstanceOEM_LCB_12x_TablePositioning_V2.wProfileNumberSet := 1;
           #InstanceOEM_LCB_12x_TablePositioning_V2.xHomingStart := TRUE;
           //Transistions
           IF #InstanceOEM_LCB_12x_TablePositioning_V2.xHomingDone THEN
               #FS.StateCases.iHoming := 52;//Executed
           ELSIF #FS.Commands.StopHoming THEN
               #FS.StateCases.iHoming := 150; //Stopping    
           END_IF;

       52: //Executing, Wait at falling edge homing sensor        
           //Actions
           #FS.CommandsActive.StartHoming := #FS.Commands.StartHoming;
           #FS.CommandsActive.StopHoming := FALSE;
           //
           #FS.Indicators.PushButtons.StartHoming := TRUE;
           #FS.Indicators.PushButtons.StopHoming := FALSE;
           #FS.Indicators.Status.IsHomed := FALSE;
           //
           #InstanceOEM_LCB_12x_TablePositioning_V2.wProfileNumberSet := 1;
           #InstanceOEM_LCB_12x_TablePositioning_V2.xHomingStart := FALSE;
           //Transistions
           IF NOT #InstanceOEM_LCB_12x_TablePositioning_V2.xHomingActive THEN
               #FS.StateCases.iHoming := 100;//Executed
           ELSIF #FS.Commands.StopHoming THEN
               #FS.StateCases.iHoming := 150; //Stopping
           END_IF;

       100: //Executed
           //Actions
           #FS.CommandsActive.StartHoming := #FS.Commands.StartHoming;
           #FS.CommandsActive.StopHoming := FALSE;
           //
           #FS.Indicators.PushButtons.StartHoming := #FS.CommandsActive.StartHoming;
           #FS.Indicators.PushButtons.StopHoming := FALSE;
           #FS.Indicators.Status.IsHomed := TRUE;
           //
           #InstanceOEM_LCB_12x_TablePositioning_V2.xHomingStart := FALSE;
           //Transistion
           IF #FS.Commands.StopHoming THEN
               #FS.StateCases.iHoming := 150; //Stopping
           ELSIF NOT #InstanceOEM_LCB_12x_TablePositioning_V2.xHomingDone THEN
               #FS.StateCases.iHoming := 150; //Stopping
           END_IF;

       150: //Stopping, Disable movement homing
           //Actions
           #FS.CommandsActive.StartHoming := FALSE;
           #FS.CommandsActive.StopHoming := #FS.Commands.StopHoming;
           //
           #FS.Indicators.PushButtons.StartHoming := FALSE;
           #FS.Indicators.PushButtons.StopHoming := TRUE;
           #FS.Indicators.Status.IsHomed := FALSE;
           //
           #InstanceOEM_LCB_12x_TablePositioning_V2.xHomingStart := FALSE;
           //Transistions
           IF #InstanceOEM_LCB_12x_TablePositioning_V2.xSpeedEqZero THEN
               #FS.StateCases.iHoming := 151; //Stopping
           END_IF;

       151: //Stopping, Reset home position
           //Actions
           #FS.CommandsActive.StartHoming := FALSE;
           #FS.CommandsActive.StopHoming := #FS.Commands.StopHoming;
           //
           #FS.Indicators.PushButtons.StartHoming := FALSE;
           #FS.Indicators.PushButtons.StopHoming := TRUE;
           #FS.Indicators.Status.IsHomed := FALSE;
           //
           #InstanceOEM_LCB_12x_TablePositioning_V2.xHomingReset := TRUE;
           //Transistions
           IF NOT #InstanceOEM_LCB_12x_TablePositioning_V2.xHomingDone THEN
               #FS.StateCases.iHoming := 152; //Stopping, Clear homing reset command
           END_IF;

       152: //Stopping, Clear homing reset command        
           //Actions
           #FS.CommandsActive.StartHoming := FALSE;
           #FS.CommandsActive.StopHoming := #FS.Commands.StopHoming;
           //
           #FS.Indicators.PushButtons.StartHoming := FALSE;
           #FS.Indicators.PushButtons.StopHoming := TRUE;
           #FS.Indicators.Status.IsHomed := FALSE;
           //
           #InstanceOEM_LCB_12x_TablePositioning_V2.xHomingReset := FALSE;
           //Transistions
           #FS.StateCases.iHoming := 0; //Stopped

   END_CASE;
END_REGION

REGION Network 16 (SCL): Functional Strategy: State Executing Automatic Position Control
   REGION Local State push service
       IF #FS.Commands.StopExecuteAutomatic AND #FS.StateCases.iExecutingAutomatic > 0 THEN
           #FS.StateCases.iExecutingAutomatic := 150; //Step pushing
       ELSIF #FS.Commands.StartExecuteAutomatic AND #FS.StateCases.iExecutingAutomatic >= 150 THEN
           #FS.StateCases.iExecutingAutomatic := 0; //Step pushing
       END_IF;

   END_REGION

   //Global Transistions handling
   IF #FS.ErrorWarning.wError <> 0 THEN
       #FS.StateCases.iExecutingAutomatic := 0; //Stopped
   END_IF;

   (*
   REGION  Autopositioning
       CASE #FS.StateCases.iExecutingAutomatic OF
           0: // Stopped
               //Actions
               #FS.CommandsActive.StartExecuteAutomatic := FALSE;
               #FS.CommandsActive.StopExecuteAutomatic := FALSE;
               //
               #FS.Indicators.PushButtons.StartExecuteAutomatic := FALSE;
               #FS.Indicators.PushButtons.StopExecuteAutomatic := FALSE;
               #FS.Indicators.Status.IsAtTargetPosSpeed := FALSE;
               //
               #InstanceOEM_LCB_12x_TablePositioning_V2.xEnablePositionTeach :=
               #InstanceOEM_LCB_12x_TablePositioning_V2.xProfileStart :=
               #InstanceOEM_LCB_12x_TablePositioning_V2.xProfileRestart :=
               #InstanceOEM_LCB_12x_TablePositioning_V2.xProfilePosStop := FALSE;
               //Transistions
               IF #FS.Commands.StartExecuteAutomatic THEN
                   #FS.StateCases.iExecutingAutomatic := 10; //Starting //20 when step 100 is not used
               END_IF;

           10: //Starting, Set profile
               //Actions
               #FS.CommandsActive.StartExecuteAutomatic := #FS.Commands.StartExecuteAutomatic;
               #FS.CommandsActive.StopExecuteAutomatic := FALSE;
               //
               #FS.Indicators.PushButtons.StartExecuteAutomatic := TRUE;
               #FS.Indicators.PushButtons.StopExecuteAutomatic := FALSE;
               #FS.Indicators.Status.IsAtTargetPosSpeed := FALSE;
               //
               #InstanceOEM_LCB_12x_TablePositioning_V2.wProfileNumberSet := 2; //Extra CPU cycle at profile2
               //Transistions
               IF TRUE THEN
                   #FS.StateCases.iExecutingAutomatic := 50; //wait for start //20 when step 100 is not used
               END_IF;

               //Used when step 100 is not used
           20: //Ready, Wait for and Execute command
               //Actions
               #FS.CommandsActive.StartExecuteAutomatic := #FS.Commands.StartExecuteAutomatic;
               #FS.CommandsActive.StopExecuteAutomatic := FALSE;
               //
               #FS.Indicators.PushButtons.StartExecuteAutomatic := TRUE;
               #FS.Indicators.PushButtons.StopExecuteAutomatic := FALSE;
               #FS.Indicators.Status.IsAtTargetPosSpeed := TRUE;
               //
               #InstanceOEM_LCB_12x_TablePositioning_V2.wProfileNumberSet := 2;
               //Transistions
               IF #FS.Commands.ExecuteLoadRecipe THEN
                   #FS.StateCases.iExecutingAutomatic := 50; //Executing
               ELSIF #FS.Commands.StopExecuteAutomatic THEN
                   #FS.StateCases.iExecutingAutomatic := 150; //Stopping
               END_IF;

           50: //Executing, Start activate new setpoint
               //Actions
               #FS.CommandsActive.StartExecuteAutomatic := #FS.Commands.StartExecuteAutomatic;
               #FS.CommandsActive.StopExecuteAutomatic := FALSE;
               //
               #FS.Indicators.PushButtons.StartExecuteAutomatic := TRUE;
               #FS.Indicators.PushButtons.StopExecuteAutomatic := FALSE;
               #FS.Indicators.Status.IsAtTargetPosSpeed := FALSE;
               //
               #InstanceOEM_LCB_12x_TablePositioning_V2.xEnablePositionTeach := FALSE;
               #InstanceOEM_LCB_12x_TablePositioning_V2.xProfileStart := FALSE;
               #InstanceOEM_LCB_12x_TablePositioning_V2.wProfileNumberSet := 2;
               //Transistions
               IF NOT #InstanceOEM_LCB_12x_TablePositioning_V2.xEnabledIsPositionTeach AND
                   NOT #InstanceOEM_LCB_12x_TablePositioning_V2.xProfileIsStarting
               THEN
                   #FS.StateCases.iExecutingAutomatic := 51; //Executing
               END_IF;

           51: //Executing, Accept new setpoint and store new setpoint to previous setpoint
               //Actions
               #FS.CommandsActive.StartExecuteAutomatic := #FS.Commands.StartExecuteAutomatic;
               #FS.CommandsActive.StopExecuteAutomatic := FALSE;
               //
               #FS.Indicators.PushButtons.StartExecuteAutomatic := TRUE;
               #FS.Indicators.PushButtons.StopExecuteAutomatic := FALSE;
               #FS.Indicators.Status.IsAtTargetPosSpeed := FALSE;
               //
               #InstanceOEM_LCB_12x_TablePositioning_V2.xEnablePositionTeach := TRUE;
               #InstanceOEM_LCB_12x_TablePositioning_V2.wProfileNumberSet := 2;
               #FS.Intern.rPreviousSpPosition_Units := #FS.Recipe.rSpPosition_Units;
               //Transistions
               IF #InstanceOEM_LCB_12x_TablePositioning_V2.xEnabledIsPositionTeach THEN
                   #FS.StateCases.iExecutingAutomatic := 52; //Executing
               END_IF;

           52: //Executing, Motion busy to new position
               //Actions
               #FS.CommandsActive.StartExecuteAutomatic := #FS.Commands.StartExecuteAutomatic;
               #FS.CommandsActive.StopExecuteAutomatic := FALSE;
               //
               #FS.Indicators.PushButtons.StartExecuteAutomatic := TRUE;
               #FS.Indicators.PushButtons.StopExecuteAutomatic := FALSE;
               #FS.Indicators.Status.IsAtTargetPosSpeed := FALSE;
               //
               #InstanceOEM_LCB_12x_TablePositioning_V2.xProfileStart := TRUE;
               #InstanceOEM_LCB_12x_TablePositioning_V2.wProfileNumberSet := 2;
               //Transistions
               IF #InstanceOEM_LCB_12x_TablePositioning_V2.xProfileIsStarting THEN
                   #FS.StateCases.iExecutingAutomatic := 53; //Executing
               END_IF;

           53: //Executing, Motion busy to new position
               //Actions
               #FS.CommandsActive.StartExecuteAutomatic := #FS.Commands.StartExecuteAutomatic;
               #FS.CommandsActive.StopExecuteAutomatic := FALSE;
               //
               #FS.Indicators.PushButtons.StartExecuteAutomatic := TRUE;
               #FS.Indicators.PushButtons.StopExecuteAutomatic := FALSE;
               #FS.Indicators.Status.IsAtTargetPosSpeed := FALSE;
               //
               #InstanceOEM_LCB_12x_TablePositioning_V2.xProfileStart := TRUE;
               #InstanceOEM_LCB_12x_TablePositioning_V2.wProfileNumberSet := 2;
               //Transistions
               IF #InstanceOEM_LCB_12x_TablePositioning_V2.xProfileDone AND
                   #InstanceOEM_LCB_12x_TablePositioning_V2.xProfileInTarget
               THEN
                   #FS.StateCases.iExecutingAutomatic := 54; //Executing,
               END_IF;

           54: //Executing, Motion busy to new position
               //Actions
               #FS.CommandsActive.StartExecuteAutomatic := #FS.Commands.StartExecuteAutomatic;
               #FS.CommandsActive.StopExecuteAutomatic := FALSE;
               //
               #FS.Indicators.PushButtons.StartExecuteAutomatic := TRUE;
               #FS.Indicators.PushButtons.StopExecuteAutomatic := FALSE;
               #FS.Indicators.Status.IsAtTargetPosSpeed := FALSE;
               //
               #InstanceOEM_LCB_12x_TablePositioning_V2.xProfileStart := FALSE;
               #InstanceOEM_LCB_12x_TablePositioning_V2.wProfileNumberSet := 2;
               //Transistions
               IF #InstanceOEM_LCB_12x_TablePositioning_V2.xProfileDone AND
                   #InstanceOEM_LCB_12x_TablePositioning_V2.xProfileInTarget
               THEN
                   #FS.StateCases.iExecutingAutomatic := 100; //Ready //20 when step 100 is not used
               END_IF;

               //Used when step 20 is not used
           100: //Executed, Wait for setpoint change
               //Actions
               #FS.CommandsActive.StartExecuteAutomatic := #FS.Commands.StartExecuteAutomatic;
               #FS.CommandsActive.StopExecuteAutomatic := FALSE;
               //
               #FS.Indicators.PushButtons.StartExecuteAutomatic := TRUE;
               #FS.Indicators.PushButtons.StopExecuteAutomatic := FALSE;
               #FS.Indicators.Status.IsAtTargetPosSpeed := TRUE;
               //
               #InstanceOEM_LCB_12x_TablePositioning_V2.wProfileNumberSet := 2;
               //Transistions
               IF #FS.Intern.rPreviousSpPosition_Units <> #FS.Recipe.rSpPosition_Units THEN
                   #FS.StateCases.iExecutingAutomatic := 50; //Executing
               ELSIF #FS.Commands.StopExecuteAutomatic THEN
                   #FS.StateCases.iExecutingAutomatic := 150; //Stopping
               END_IF;

           150: //Stopping, wait till motion is in stilstand
               //Actions
               #FS.CommandsActive.StartExecuteAutomatic := FALSE;
               #FS.CommandsActive.StopExecuteAutomatic := #FS.Commands.StopExecuteAutomatic;
               //
               #FS.Indicators.PushButtons.StartExecuteAutomatic := FALSE;
               #FS.Indicators.PushButtons.StopExecuteAutomatic := TRUE;
               #FS.Indicators.Status.IsAtTargetPosSpeed := FALSE;
               //
               #InstanceOEM_LCB_12x_TablePositioning_V2.xEnablePositionTeach :=
               #InstanceOEM_LCB_12x_TablePositioning_V2.xProfileStart :=
               #InstanceOEM_LCB_12x_TablePositioning_V2.xProfileRestart := FALSE;

               #InstanceOEM_LCB_12x_TablePositioning_V2.xProfilePosStop := TRUE;
               #InstanceOEM_LCB_12x_TablePositioning_V2.wProfileNumberSet := 2;
               //Transistions
               IF #InstanceOEM_LCB_12x_TablePositioning_V2.xSpeedEqZero THEN
                   #FS.StateCases.iExecutingAutomatic := 151; //Stopping, 
               END_IF;

           151: //Stopping, ending
               //Actions
               #FS.CommandsActive.StartExecuteAutomatic := FALSE;
               #FS.CommandsActive.StopExecuteAutomatic := #FS.Commands.StopExecuteAutomatic;
               //
               #FS.Indicators.PushButtons.StartExecuteAutomatic := FALSE;
               #FS.Indicators.PushButtons.StopExecuteAutomatic := TRUE;
               #FS.Indicators.Status.IsAtTargetPosSpeed := FALSE;
               //
               #InstanceOEM_LCB_12x_TablePositioning_V2.xProfilePosStop := FALSE;
               //Transistions
               IF TRUE THEN
                   #FS.StateCases.iExecutingAutomatic := 0; //Stopped
               END_IF;
       END_CASE;
   END_REGION
   *)

   REGION ExecuteLoadRecipe
       CASE #FS.StateCases.iExecutingAutomatic OF
           0: // Stopped
               //Actions
               #FS.CommandsActive.StartExecuteAutomatic := FALSE;
               #FS.CommandsActive.StopExecuteAutomatic := FALSE;
               //
               #FS.Indicators.PushButtons.StartExecuteAutomatic := FALSE;
               #FS.Indicators.PushButtons.StopExecuteAutomatic := FALSE;
               #FS.Indicators.PushButtons.ExecuteLoadRecipe := FALSE;
               #FS.Indicators.Status.IsAtTargetPosSpeed := FALSE;
               //
               #InstanceOEM_LCB_12x_TablePositioning_V2.xEnablePositionTeach :=
               #InstanceOEM_LCB_12x_TablePositioning_V2.xProfileStart :=
               #InstanceOEM_LCB_12x_TablePositioning_V2.xProfileRestart :=
               #InstanceOEM_LCB_12x_TablePositioning_V2.xProfilePosStop := FALSE;
               //Transistions
               IF #FS.Commands.StartExecuteAutomatic THEN
                   #FS.StateCases.iExecutingAutomatic := 10; //Starting
               END_IF;

           10: //Starting, Set profile
               //Actions
               #FS.CommandsActive.StartExecuteAutomatic := #FS.Commands.StartExecuteAutomatic;
               #FS.CommandsActive.StopExecuteAutomatic := FALSE;
               //
               #FS.Indicators.PushButtons.StartExecuteAutomatic := TRUE;
               #FS.Indicators.PushButtons.StopExecuteAutomatic := FALSE;
               #FS.Indicators.PushButtons.ExecuteLoadRecipe := #FS.Commands.ExecuteLoadRecipe;
               #FS.Indicators.Status.IsAtTargetPosSpeed := FALSE;
               //
               #InstanceOEM_LCB_12x_TablePositioning_V2.wProfileNumberSet := 2; //Extra CPU cycle at profile2
               //Transistions
               IF TRUE THEN
                   #FS.StateCases.iExecutingAutomatic := 20; //wait for start
               END_IF;

           20: //Ready, Wait for and Execute command
               //Actions
               #FS.CommandsActive.StartExecuteAutomatic := #FS.Commands.StartExecuteAutomatic;
               #FS.CommandsActive.StopExecuteAutomatic := FALSE;
               //
               #FS.Indicators.PushButtons.StartExecuteAutomatic := TRUE;
               #FS.Indicators.PushButtons.StopExecuteAutomatic := FALSE;
               #FS.Indicators.PushButtons.ExecuteLoadRecipe := #FS.Commands.ExecuteLoadRecipe;
               #FS.Indicators.Status.IsAtTargetPosSpeed := TRUE;
               //
               #InstanceOEM_LCB_12x_TablePositioning_V2.wProfileNumberSet := 2;
               //Transistions
               IF #FS.Commands.ExecuteLoadRecipe THEN
                   #FS.StateCases.iExecutingAutomatic := 50; //Executing
               ELSIF #FS.Commands.StopExecuteAutomatic THEN
                   #FS.StateCases.iExecutingAutomatic := 150; //Stopping
               END_IF;

           50: //Executing, Start activate new setpoint
               //Actions
               #FS.CommandsActive.StartExecuteAutomatic := #FS.Commands.StartExecuteAutomatic;
               #FS.CommandsActive.StopExecuteAutomatic := FALSE;
               //
               #FS.Indicators.PushButtons.StartExecuteAutomatic := TRUE;
               #FS.Indicators.PushButtons.StopExecuteAutomatic := FALSE;
               #FS.Indicators.PushButtons.ExecuteLoadRecipe := #FS.Commands.ExecuteLoadRecipe;
               #FS.Indicators.Status.IsAtTargetPosSpeed := FALSE;
               //
               #InstanceOEM_LCB_12x_TablePositioning_V2.xEnablePositionTeach := FALSE;
               #InstanceOEM_LCB_12x_TablePositioning_V2.xProfileStart := FALSE;
               #InstanceOEM_LCB_12x_TablePositioning_V2.wProfileNumberSet := 2;
               //Transistions
               IF NOT #InstanceOEM_LCB_12x_TablePositioning_V2.xEnabledIsPositionTeach AND
                   NOT #InstanceOEM_LCB_12x_TablePositioning_V2.xProfileIsStarting
               THEN
                   #FS.StateCases.iExecutingAutomatic := 51; //Executing
               END_IF;

           51: //Executing, Accept new setpoint and store new setpoint to previous setpoint
               //Actions
               #FS.CommandsActive.StartExecuteAutomatic := #FS.Commands.StartExecuteAutomatic;
               #FS.CommandsActive.StopExecuteAutomatic := FALSE;
               //
               #FS.Indicators.PushButtons.StartExecuteAutomatic := TRUE;
               #FS.Indicators.PushButtons.StopExecuteAutomatic := FALSE;
               #FS.Indicators.PushButtons.ExecuteLoadRecipe := #FS.Commands.ExecuteLoadRecipe;
               #FS.Indicators.Status.IsAtTargetPosSpeed := FALSE;
               //
               #InstanceOEM_LCB_12x_TablePositioning_V2.xEnablePositionTeach := TRUE;
               #InstanceOEM_LCB_12x_TablePositioning_V2.wProfileNumberSet := 2;
               #FS.Intern.rPreviousSpPosition_Units := #FS.Recipe.rSpPosition_Units;
               //Transistions
               IF #InstanceOEM_LCB_12x_TablePositioning_V2.xEnabledIsPositionTeach THEN
                   #FS.StateCases.iExecutingAutomatic := 52; //Executing
               END_IF;

           52: //Executing, Motion busy to new position
               //Actions
               #FS.CommandsActive.StartExecuteAutomatic := #FS.Commands.StartExecuteAutomatic;
               #FS.CommandsActive.StopExecuteAutomatic := FALSE;
               //
               #FS.Indicators.PushButtons.StartExecuteAutomatic := TRUE;
               #FS.Indicators.PushButtons.StopExecuteAutomatic := FALSE;
               #FS.Indicators.PushButtons.ExecuteLoadRecipe := #FS.Commands.ExecuteLoadRecipe;
               #FS.Indicators.Status.IsAtTargetPosSpeed := FALSE;
               //
               #InstanceOEM_LCB_12x_TablePositioning_V2.xProfileStart := TRUE;
               #InstanceOEM_LCB_12x_TablePositioning_V2.wProfileNumberSet := 2;
               //Transistions
               IF #InstanceOEM_LCB_12x_TablePositioning_V2.xProfileIsStarting THEN
                   #FS.StateCases.iExecutingAutomatic := 53; //Executing
               END_IF;

           53: //Executing, Motion busy to new position
               //Actions
               #FS.CommandsActive.StartExecuteAutomatic := #FS.Commands.StartExecuteAutomatic;
               #FS.CommandsActive.StopExecuteAutomatic := FALSE;
               //
               #FS.Indicators.PushButtons.StartExecuteAutomatic := TRUE;
               #FS.Indicators.PushButtons.StopExecuteAutomatic := FALSE;
               #FS.Indicators.PushButtons.ExecuteLoadRecipe := #FS.Commands.ExecuteLoadRecipe;
               #FS.Indicators.Status.IsAtTargetPosSpeed := FALSE;
               //
               #InstanceOEM_LCB_12x_TablePositioning_V2.xProfileStart := TRUE;
               #InstanceOEM_LCB_12x_TablePositioning_V2.wProfileNumberSet := 2;
               //Transistions
               IF #InstanceOEM_LCB_12x_TablePositioning_V2.xProfileDone AND
                   #InstanceOEM_LCB_12x_TablePositioning_V2.xProfileInTarget
               THEN
                   #FS.StateCases.iExecutingAutomatic := 54; //Executing, 
               END_IF;

           54: //Executing, Motion busy to new position
               //Actions
               #FS.CommandsActive.StartExecuteAutomatic := #FS.Commands.StartExecuteAutomatic;
               #FS.CommandsActive.StopExecuteAutomatic := FALSE;
               //
               #FS.Indicators.PushButtons.StartExecuteAutomatic := TRUE;
               #FS.Indicators.PushButtons.StopExecuteAutomatic := FALSE;
               #FS.Indicators.PushButtons.ExecuteLoadRecipe := #FS.Commands.ExecuteLoadRecipe;
               #FS.Indicators.Status.IsAtTargetPosSpeed := FALSE;
               //
               #InstanceOEM_LCB_12x_TablePositioning_V2.xProfileStart := FALSE;
               #InstanceOEM_LCB_12x_TablePositioning_V2.wProfileNumberSet := 2;
               //Transistions
               IF #InstanceOEM_LCB_12x_TablePositioning_V2.xProfileDone AND
                   #InstanceOEM_LCB_12x_TablePositioning_V2.xProfileInTarget
               THEN
                   #FS.StateCases.iExecutingAutomatic := 100; //Executed
               END_IF;

           100: //Executed, Wait for setpoint change
               //Actions
               #FS.CommandsActive.StartExecuteAutomatic := #FS.Commands.StartExecuteAutomatic;
               #FS.CommandsActive.StopExecuteAutomatic := FALSE;
               //
               #FS.Indicators.PushButtons.StartExecuteAutomatic := TRUE;
               #FS.Indicators.PushButtons.StopExecuteAutomatic := FALSE;
               #FS.Indicators.PushButtons.ExecuteLoadRecipe := #FS.Commands.ExecuteLoadRecipe;
               #FS.Indicators.Status.IsAtTargetPosSpeed := TRUE;
               //
               #InstanceOEM_LCB_12x_TablePositioning_V2.wProfileNumberSet := 2;
               //Transistions
               IF #FS.Intern.rPreviousSpPosition_Units <> #FS.Recipe.rSpPosition_Units THEN
                   #FS.StateCases.iExecutingAutomatic := 20; //Ready
               ELSIF #FS.Commands.StopExecuteAutomatic THEN
                   #FS.StateCases.iExecutingAutomatic := 150; //Stopping
               END_IF;

           150: //Stopping, wait till motion is in stilstand
               //Actions
               #FS.CommandsActive.StartExecuteAutomatic := FALSE;
               #FS.CommandsActive.StopExecuteAutomatic := #FS.Commands.StopExecuteAutomatic;
               //
               #FS.Indicators.PushButtons.StartExecuteAutomatic := FALSE;
               #FS.Indicators.PushButtons.StopExecuteAutomatic := TRUE;
               #FS.Indicators.PushButtons.ExecuteLoadRecipe := #FS.Commands.ExecuteLoadRecipe;
               #FS.Indicators.Status.IsAtTargetPosSpeed := FALSE;
               //
               #InstanceOEM_LCB_12x_TablePositioning_V2.xEnablePositionTeach :=
               #InstanceOEM_LCB_12x_TablePositioning_V2.xProfileStart :=
               #InstanceOEM_LCB_12x_TablePositioning_V2.xProfileRestart := FALSE;

               #InstanceOEM_LCB_12x_TablePositioning_V2.xProfilePosStop := TRUE;
               #InstanceOEM_LCB_12x_TablePositioning_V2.wProfileNumberSet := 2;
               //Transistions
               IF #InstanceOEM_LCB_12x_TablePositioning_V2.xSpeedEqZero THEN
                   #FS.StateCases.iExecutingAutomatic := 151; //Stopping, 
               END_IF;

           151: //Stopping, ending
               //Actions
               #FS.CommandsActive.StartExecuteAutomatic := FALSE;
               #FS.CommandsActive.StopExecuteAutomatic := #FS.Commands.StopExecuteAutomatic;
               //
               #FS.Indicators.PushButtons.StartExecuteAutomatic := FALSE;
               #FS.Indicators.PushButtons.StopExecuteAutomatic := TRUE;
               #FS.Indicators.PushButtons.ExecuteLoadRecipe := #FS.Commands.ExecuteLoadRecipe;
               #FS.Indicators.Status.IsAtTargetPosSpeed := FALSE;
               //
               #InstanceOEM_LCB_12x_TablePositioning_V2.xProfilePosStop := FALSE;
               //Transistions
               IF TRUE THEN
                   #FS.StateCases.iExecutingAutomatic := 0; //Stopped
               END_IF;
       END_CASE;
   END_REGION
END_REGION

REGION Network 17 (SCL): Functional Strategy: SingleStep Mode--> Restore actual State cases
   IF #FM.ModeActual = 5 (*SingleStep Mode*)THEN
       IF #FS.Commands.PbSingleStep THEN
           #FS.StateCases := #FS.StateCases;
       ELSE
           #FS.StateCases := #FS.StateCasesPrevious;
       END_IF;
   END_IF;
END_REGION

REGION Network 18: Functional Strategy: OEM SetAxisData Application
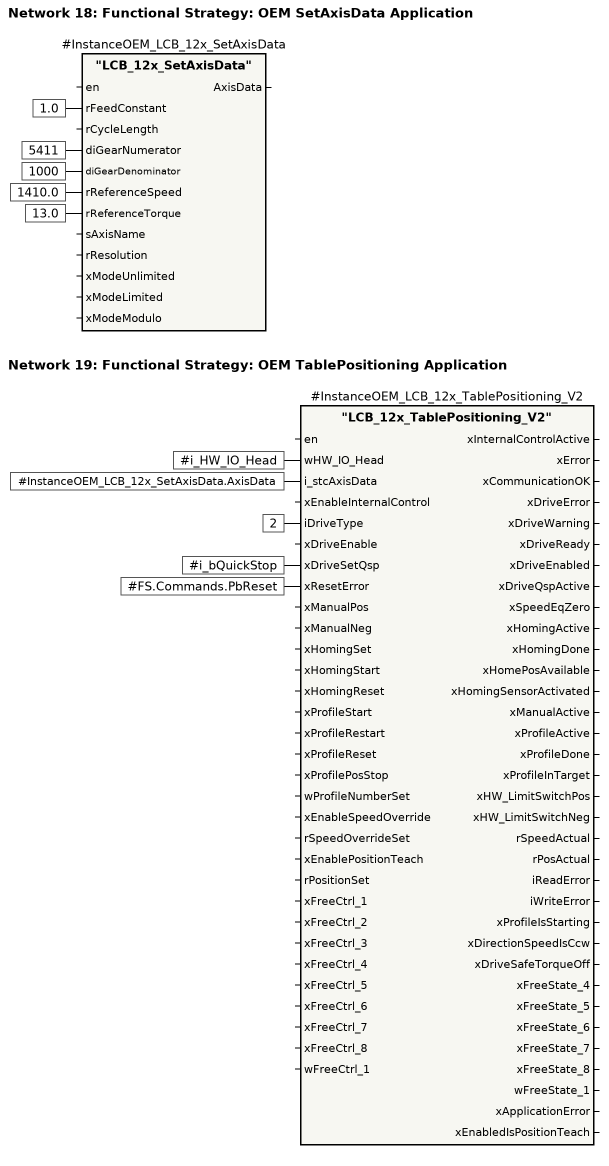
   #InstanceOEM_LCB_12x_SetAxisData(rFeedConstant := 1.0,   // "LCB_12x_SetAxisData"
                           diGearNumerator := 5411,
                           diGearDenominator := 1000,
                           rReferenceSpeed := 1410.0,
                           rReferenceTorque := 13.0);
END_REGION

REGION Network 19: Functional Strategy: OEM TablePositioning Application
   #InstanceOEM_LCB_12x_TablePositioning_V2(wHW_IO_Head := #i_HW_IO_Head,   // "LCB_12x_TablePositioning_V2"
                           i_stcAxisData := #InstanceOEM_LCB_12x_SetAxisData.AxisData,
                           iDriveType := 2,
                           xDriveSetQsp := #i_bQuickStop,
                           xResetError := #FS.Commands.PbReset);
END_REGION

REGION Network 20 (SCL): Functional strategy: OEM Range Process values
   IF #InstanceOEM_LCB_12x_TablePositioning_V2.xHomingDone THEN
       #FS.ProcessValues.rPvPosition_Units :=
           #InstanceOEM_LCB_12x_TablePositioning_V2.rPosActual +
           #FS.Settings.rSpLimitH_Units -
           #FS.Settings.rSpPositionOffset_Units;
   ELSE
       #FS.ProcessValues.rPvPosition_Units := 3.402823e+38;
   END_IF;
END_REGION

REGION Network 21 (SCL): Functional Strategy: Enable/ Disable Error/Warning release
   // Enable release error / warning 
   IF #FS.Commands.EnableReleaseErrorWarning THEN
       #FS.Intern.ErrorWarningReleased := true;
   END_IF;

   // Disable release error / warning 
   IF #FS.Commands.DisableReleaseErrorWarning THEN
       #FS.Intern.ErrorWarningReleased := false;
   END_IF;
END_REGION

REGION Network 22 (SCL): Functional Strategy: Error Warning Module
   REGION #FS.ErrorWarningModule.wError
       IF NOT #FS.Intern.ErrorWarningReleased THEN
           #FS.ErrorWarningModule.wError := 0;
           #FS.ErrorWarningModule.bErrorTripped := 0;
       ELSIF #FS.Intern.ErrorWarningReleased THEN
           #FS.ErrorWarningModule.wError.%X0 := false;
           #FS.ErrorWarningModule.wError.%X1 := FALSE;
           #FS.ErrorWarningModule.wError.%X2 := FALSE;
           #FS.ErrorWarningModule.wError.%X3 := FALSE;
           #FS.ErrorWarningModule.wError.%X4 := FALSE;
           #FS.ErrorWarningModule.wError.%X5 := FALSE;
           #FS.ErrorWarningModule.wError.%X6 := FALSE;
           #FS.ErrorWarningModule.wError.%X7 := FALSE;
           #FS.ErrorWarningModule.wError.%X8 := FALSE;
           #FS.ErrorWarningModule.wError.%X9 := FALSE;
           #FS.ErrorWarningModule.wError.%X10 := FALSE;
           #FS.ErrorWarningModule.wError.%X11 := FALSE;
           #FS.ErrorWarningModule.wError.%X12 := FALSE;
           #FS.ErrorWarningModule.wError.%X13 := FALSE;
           #FS.ErrorWarningModule.wError.%X14 := FALSE;
           #FS.ErrorWarningModule.wError.%X15 := FALSE;
           //
           #FS.ErrorWarningModule.bErrorTripped := #FS.ErrorWarningModule.wError > 0;
       END_IF;
   END_REGION

   REGION #FS.ErrorWarningModule.wWarning
       IF NOT #FS.Intern.ErrorWarningReleased THEN
           #FS.ErrorWarningModule.wWarning := 0;
           #FS.ErrorWarningModule.bWarningTripped := 0;
       ELSIF #FS.Intern.ErrorWarningReleased THEN
           #FS.ErrorWarningModule.wWarning.%X0 := FALSE;
           #FS.ErrorWarningModule.wWarning.%X1 := FALSE;
           #FS.ErrorWarningModule.wWarning.%X2 := FALSE;
           #FS.ErrorWarningModule.wWarning.%X3 := FALSE;
           #FS.ErrorWarningModule.wWarning.%X4 := FALSE;
           #FS.ErrorWarningModule.wWarning.%X5 := FALSE;
           #FS.ErrorWarningModule.wWarning.%X6 := FALSE;
           #FS.ErrorWarningModule.wWarning.%X7 := FALSE;
           #FS.ErrorWarningModule.wWarning.%X8 := FALSE;
           #FS.ErrorWarningModule.wWarning.%X9 := FALSE;
           #FS.ErrorWarningModule.wWarning.%X10 := FALSE;
           #FS.ErrorWarningModule.wWarning.%X11 := FALSE;
           #FS.ErrorWarningModule.wWarning.%X12 := FALSE;
           #FS.ErrorWarningModule.wWarning.%X13 := FALSE;
           #FS.ErrorWarningModule.wWarning.%X14 := FALSE;
           #FS.ErrorWarningModule.wWarning.%X15 := FALSE;
           //
           #FS.ErrorWarningModule.bWarningTripped := #FS.ErrorWarningModule.wWarning> 0;
       END_IF;
   END_REGION
END_REGION

REGION Network 23 (SCL): Functional Strategy: Error Warning OEM device
   REGION #FS.ErrorWarning.wError
       IF NOT #FS.Intern.ErrorWarningReleased THEN
           #FS.ErrorWarning.wError := 0;
           #FS.ErrorWarning.bErrorTripped := 0;
       ELSIF #InstanceOEM_LCB_12x_TablePositioning_V2.iReadError <> 0 THEN
           #FS.ErrorWarning.wError := INT_TO_WORD(#InstanceOEM_LCB_12x_TablePositioning_V2.iReadError);//Mapping drive communication reading data error
       ELSIF #InstanceOEM_LCB_12x_TablePositioning_V2.iWriteError <> 0 THEN
           #FS.ErrorWarning.wError := INT_TO_WORD(#InstanceOEM_LCB_12x_TablePositioning_V2.iWriteError);//Mapping drive communication reading data error
       ELSE
           #FS.ErrorWarning.wError.%X0 := #InstanceOEM_LCB_12x_TablePositioning_V2.xError;
           #FS.ErrorWarning.wError.%X1 := NOT #InstanceOEM_LCB_12x_TablePositioning_V2.xCommunicationOK;
           #FS.ErrorWarning.wError.%X2 := #InstanceOEM_LCB_12x_TablePositioning_V2.xDriveError;
           #FS.ErrorWarning.wError.%X3 := #InstanceOEM_LCB_12x_TablePositioning_V2.xDriveQspActive AND NOT #i_bQuickStop;
           #FS.ErrorWarning.wError.%X4 := #InstanceOEM_LCB_12x_TablePositioning_V2.xApplicationError;
           #FS.ErrorWarning.wError.%X5 := #InstanceOEM_LCB_12x_TablePositioning_V2.xDriveSafeTorqueOff;
           #FS.ErrorWarning.wError.%X6 := FALSE;
           #FS.ErrorWarning.wError.%X7 := FALSE;
           #FS.ErrorWarning.wError.%X8 := FALSE;
           #FS.ErrorWarning.wError.%X9 := FALSE;
           #FS.ErrorWarning.wError.%X10 := FALSE;
           #FS.ErrorWarning.wError.%X11 := FALSE;
           #FS.ErrorWarning.wError.%X12 := FALSE;
           #FS.ErrorWarning.wError.%X13 := FALSE;
           #FS.ErrorWarning.wError.%X14 := FALSE;
           #FS.ErrorWarning.wError.%X15 := FALSE;
           //
           #FS.ErrorWarning.bErrorTripped := #FS.ErrorWarning.wError > 0;
       END_IF;
   END_REGION

   REGION #FS.ErrorWarning.wWarning
       IF NOT #FS.Intern.ErrorWarningReleased THEN
           #FS.ErrorWarning.wWarning := 0;
           #FS.ErrorWarning.bWarningTripped := 0;
       ELSIF #FS.Intern.ErrorWarningReleased THEN
           #FS.ErrorWarning.wWarning.%X0 := #InstanceOEM_LCB_12x_TablePositioning_V2.xDriveWarning;
           #FS.ErrorWarning.wWarning.%X1 := #InstanceOEM_LCB_12x_TablePositioning_V2.xHW_LimitSwitchNeg;
           #FS.ErrorWarning.wWarning.%X2 := #InstanceOEM_LCB_12x_TablePositioning_V2.xHW_LimitSwitchPos;
           #FS.ErrorWarning.wWarning.%X3 := FALSE;
           #FS.ErrorWarning.wWarning.%X4 := FALSE;
           #FS.ErrorWarning.wWarning.%X5 := FALSE;
           #FS.ErrorWarning.wWarning.%X6 := FALSE;
           #FS.ErrorWarning.wWarning.%X7 := FALSE;
           #FS.ErrorWarning.wWarning.%X8 := FALSE;
           #FS.ErrorWarning.wWarning.%X9 := FALSE;
           #FS.ErrorWarning.wWarning.%X10 := FALSE;
           #FS.ErrorWarning.wWarning.%X11 := FALSE;
           #FS.ErrorWarning.wWarning.%X12 := FALSE;
           #FS.ErrorWarning.wWarning.%X13 := FALSE;
           #FS.ErrorWarning.wWarning.%X14 := FALSE;
           #FS.ErrorWarning.wWarning.%X15 := FALSE;
           //
           #FS.ErrorWarning.bWarningTripped := #FS.ErrorWarning.wWarning> 0;
       END_IF;
   END_REGION
END_REGION

REGION Network 24 (SCL): Functional Strategy: State Error (Error-ID Mapping at 32bit)
   REGION Explaining structure of Error-ID
   (*
   ModuleErrorID = 32bit Integer as status output
   ErrorModuleID = 32 bit Word as value 0..4.294.967.295

   31,30,29,28,27,26,25,24,23,22,21,20,19,18,17,16,15,14,13,12,11,10,9,8,7,6,5,4,3,2,1,0 
                                                   15,14,13,12,11,10,9,8,7,6,5,4,3,2,1,0 
                                                   Error ID = 16 bit Word as value 0..65635 Example: Dc bus undervoltage
                      25,24,23,22,21,20,19,18,17,16
                      Error subject area  = 10 bit Word as value 0..65635 Example: Supply voltage, Temperature, Device hardware defective
   31,30,29,28,27,26
   Error location area = 6 bit Word as value 0..63 Example: TopDosingRoll Temperature control, BottomRoll Drive
   *)
   END_REGION

   REGION Declare Error Mapping area's coded in  32BitID
   (*Declare Error location area
   1= Error subject area Module:  no module errors defined yet
   2= Error subject area Drive Communication:
   3= Error subject area Drive Lenze ID:
   *)
       #FS.ErrorWarning.iAdressAreaSize := 3; // Set the count of Error locations 

   (*LocationArea1 SubjectArea xx:
   1= Error Word
   2= Warning Word
   *)
   (*LocationArea2 SubjectArea xx:
   1= #InstanceOEM_LCB_12x_TablePositioning_V2.iReadError
   2= #InstanceOEM_LCB_12x_TablePositioning_V2.iWriteError
   *)
   (*LocationArea3 SubjectArea xx:
   NOT provided jet in the communcation data packet. 
   The Lenze drive is ready TO use but is NOT couple at the communication data TO PLC
   SubjectArea is Mapped inside the 32bit Lenze Error ID Double word
   *)
   END_REGION

   IF NOT #FS.Intern.ErrorWarningReleased THEN
       #FS.Intern.ErrorWarning.wErrorLocationArea := 0;
       #FS.Intern.ErrorWarning.wErrorSubjectArea := 0;
       #FS.Intern.ErrorWarning.wErrorID := 0;
   ELSIF #FS.Intern.ErrorWarningReleased THEN

       //Handling first trigger Error or Warning
       IF #FS.StateCases.iError = 0 OR //0= No error or warning active
           #FS.StateCases.iError >= 500  //warning is active. If Warning is active an Error must be detected as ID
       THEN
           IF #FS.ErrorWarningModule.wError <> 0 THEN
               #FS.StateCases.iError := 10;//Mapping local module wError
           ELSIF #FS.ErrorWarning.wError <> 0 THEN
               #FS.StateCases.iError := 20;//Mapping drive communication reading data error
           (*ELSIF #InstanceOEM_LCB_12x_TablePositioning_V2.iWriteError <> 0 THEN
               #FS.StateCases.iError := 30;////Mapping drive communication writing data error  *)            
           (*  ELSIF #InstanceOEM_LCB_12x_TablePositioning_V2.dwErrorID <> 0 THEN
                 #FS.State.iError := 40;//Mapping drive warning or error    *)
           ELSIF #FS.ErrorWarning.wWarning <> 0 AND
                   #FS.StateCases.iError < 500 THEN //Mapping warning only at the first trigger
               #FS.StateCases.iError := 500;//Mapping wWarning     
           END_IF;
       END_IF;

       CASE #FS.StateCases.iError OF //Error Warning Mapping to ID
       0: // No Error, Area mapping handling
           //Actions
           #FS.ErrorWarning.diModuleErrorID := 0;
           //Transistions
           (*
               This transistion is handeld outside the case.
           *)
       10: // Mapping wError
           // Actions
           #FS.Intern.ErrorWarning.wErrorLocationArea := 1 + INT_TO_WORD(#CD.iStartAreaAdressErrorID);
           #FS.Intern.ErrorWarning.wErrorSubjectArea := 1;
           #FS.Intern.ErrorWarning.wErrorID := #FS.ErrorWarningModule.wError;
           #FS.Intern.ErrorWarning.bErrorTripped := #FS.ErrorWarningModule.bErrorTripped;
           #FS.Intern.ErrorWarning.bWarningTripped := #FS.ErrorWarningModule.bWarningTripped;
           //Transistions
           IF TRUE THEN
               #FS.StateCases.iError := 11; //Next step
           END_IF;
       11: //Mapping LocationArea1 SubjectArea1
           //Transistions
           IF #FS.ErrorWarningModule.wError = 0 THEN
               #FS.StateCases.iError := 0; //No Error
           END_IF;

   (*Mapping LocationArea1 SubjectArea1*)        
       20: //Mapping LocationArea1 SubjectArea1
           //Actions
           #FS.Intern.ErrorWarning.wErrorLocationArea := 1 + INT_TO_WORD(#CD.iStartAreaAdressErrorID);
           #FS.Intern.ErrorWarning.wErrorSubjectArea := 2;
           #FS.Intern.ErrorWarning.wErrorID := #FS.ErrorWarning.wError;
           #FS.Intern.ErrorWarning.bErrorTripped := #FS.ErrorWarning.bErrorTripped;
           #FS.Intern.ErrorWarning.bWarningTripped := #FS.ErrorWarning.bWarningTripped;
           //Transistions
           IF TRUE THEN
               #FS.StateCases.iError := 21; //Next step
           END_IF;
       21: //Mapping LocationArea1 SubjectArea1
           //Transistions
           IF #FS.ErrorWarning.wError = 0 THEN
               #FS.StateCases.iError := 0; //No Error
           END_IF;

   (*Mapping LocationArea2 SubjectArea1*)        
       30: //Mapping LocationArea2 SubjectArea1
           //Actions
           #FS.Intern.ErrorWarning.wErrorLocationArea := 2 + INT_TO_WORD(#CD.iStartAreaAdressErrorID);
           (*#FS.Intern.ErrorWarning.wErrorSubjectArea := 2;
           #FS.Intern.ErrorWarning.wErrorID := INT_TO_WORD(#InstanceOEM_LCB_12x_TablePositioning_V2.iReadError);*)
           //Transistions
           IF TRUE THEN
               #FS.StateCases.iError := 31; //Next step
           END_IF;
       31: //Mapping LocationArea2 SubjectArea1
           //Transistions
           //IF #InstanceOEM_LCB_12x_TablePositioning_V2.iReadError = 0 THEN
               #FS.StateCases.iError := 0; //No Error
           //END_IF;

   (*Mapping LocationArea3 SubjectArea xx*)        
       40: //Mapping LocationArea3 SubjectArea xx
           //Actions
           (*wErrorLocationArea*)
           #FS.Intern.ErrorWarning.wErrorLocationArea := 3 + INT_TO_WORD(#CD.iStartAreaAdressErrorID);

           (* wErrorSubjectArea
           #FS.Intern.wErrorSubjectArea.%X0    :=  #InstanceOEM_LCB_12x_TablePositioning_V2.dwErrorID.X16
           #FS.Intern.wErrorSubjectArea.%X1    :=  #InstanceOEM_LCB_12x_TablePositioning_V2.dwErrorID.X17
           #FS.Intern.wErrorSubjectArea.%X2    :=  #InstanceOEM_LCB_12x_TablePositioning_V2.dwErrorID.X18
           #FS.Intern.wErrorSubjectArea.%X3    :=  #InstanceOEM_LCB_12x_TablePositioning_V2.dwErrorID.X19
           #FS.Intern.wErrorSubjectArea.%X4    :=  #InstanceOEM_LCB_12x_TablePositioning_V2.dwErrorID.X20
           #FS.Intern.wErrorSubjectArea.%X5    :=  #InstanceOEM_LCB_12x_TablePositioning_V2.dwErrorID.X21
           #FS.Intern.wErrorSubjectArea.%X6    :=  #InstanceOEM_LCB_12x_TablePositioning_V2.dwErrorID.X22
           #FS.Intern.wErrorSubjectArea.%X7    :=  #InstanceOEM_LCB_12x_TablePositioning_V2.dwErrorID.X23
           #FS.Intern.wErrorSubjectArea.%X8    :=  #InstanceOEM_LCB_12x_TablePositioning_V2.dwErrorID.X24
           #FS.Intern.wErrorSubjectArea.%X9    :=  #InstanceOEM_LCB_12x_TablePositioning_V2.dwErrorID.X25
           *)

           (*wErrorID
           #FS.Intern.wErrorID.%X0 :=  #InstanceOEM_LCB_12x_TablePositioning_V2.dwErrorID.X0
           #FS.Intern.wErrorID.%X1 :=  #InstanceOEM_LCB_12x_TablePositioning_V2.dwErrorID.X1
           #FS.Intern.wErrorID.%X2 :=  #InstanceOEM_LCB_12x_TablePositioning_V2.dwErrorID.X2
           #FS.Intern.wErrorID.%X3 :=  #InstanceOEM_LCB_12x_TablePositioning_V2.dwErrorID.X3
           #FS.Intern.wErrorID.%X4 :=  #InstanceOEM_LCB_12x_TablePositioning_V2.dwErrorID.X4
           #FS.Intern.wErrorID.%X5 :=  #InstanceOEM_LCB_12x_TablePositioning_V2.dwErrorID.X5
           #FS.Intern.wErrorID.%X6 :=  #InstanceOEM_LCB_12x_TablePositioning_V2.dwErrorID.X6
           #FS.Intern.wErrorID.%X7 :=  #InstanceOEM_LCB_12x_TablePositioning_V2.dwErrorID.X7
           #FS.Intern.wErrorID.%X8 :=  #InstanceOEM_LCB_12x_TablePositioning_V2.dwErrorID.X8
           #FS.Intern.wErrorID.%X9 :=  #InstanceOEM_LCB_12x_TablePositioning_V2.dwErrorID.X9
           #FS.Intern.wErrorID.%X10    :=  #InstanceOEM_LCB_12x_TablePositioning_V2.dwErrorID.X10
           #FS.Intern.wErrorID.%X11    :=  #InstanceOEM_LCB_12x_TablePositioning_V2.dwErrorID.X11
           #FS.Intern.wErrorID.%X12    :=  #InstanceOEM_LCB_12x_TablePositioning_V2.dwErrorID.X12
           #FS.Intern.wErrorID.%X13    :=  #InstanceOEM_LCB_12x_TablePositioning_V2.dwErrorID.X13
           #FS.Intern.wErrorID.%X14    :=  #InstanceOEM_LCB_12x_TablePositioning_V2.dwErrorID.X14
           #FS.Intern.wErrorID.%X15    :=  #InstanceOEM_LCB_12x_TablePositioning_V2.dwErrorID.X15
           *)

           //Transistions
           IF TRUE THEN
               #FS.StateCases.iError := 41; //Next step
           END_IF;

       41: //Mapping LocationArea3 SubjectArea xx
           //Transistions
         //  IF #InstanceOEM_LCB_12x_TablePositioning_V2.dwErrorID = 0 THEN
               #FS.StateCases.iError := 0; //No Error
         //  END_IF;

   (*//Mapping LocationArea1 SubjectArea2*)
       500: //Mapping LocationArea1 SubjectArea2
           //Actions
           #FS.Intern.ErrorWarning.wErrorLocationArea := 1 + INT_TO_WORD(#CD.iStartAreaAdressErrorID);
           #FS.Intern.ErrorWarning.wErrorSubjectArea := 2;
           #FS.Intern.ErrorWarning.wErrorID := #FS.ErrorWarning.wWarning;
           //Transistions
           IF TRUE THEN
               #FS.StateCases.iError := 501; //Next step
           END_IF;
       501: //Mapping LocationArea1 SubjectArea2
           //Transistions
           IF #FS.ErrorWarning.wWarning = 0 THEN
               #FS.StateCases.iError := 0; //No Error
           END_IF;

   END_CASE; //32 bit Error-ID mapping
   END_IF;
END_REGION

REGION Network 25 (SCL): Functional Strategy: Mapping Outputs
   #q_bDriveIEnableRfr := #FS.Outputs.bDriveInhibitTerminal;
END_REGION

REGION Network 26 (SCL): Functional Strategy: Mapping to SD
   #SD.bRFR := #FS.StateCases.iModule = 70;//ReadyHomed
   #SD.bExecuting := #FS.StateCases.iModule = 80; //Executing
   #SD.bRecipeAccepted := #FS.Recipe = #CD.Recipe; //Local recipe FS must is equal at Control data recipe
   #SD.CommandsActivated := #FS.CommandsActive;

   REGION ErrorWarning
       #SD.ErrorWarning.bErrorTripped := #FS.ErrorWarning.bErrorTripped;
       #SD.ErrorWarning.bWarningTripped := #FS.ErrorWarning.bWarningTripped;
       #SD.ErrorWarning.iAdressAreaSize := #FS.ErrorWarning.iAdressAreaSize;
       #SD.ErrorWarning.diModuleErrorID := DWORD_TO_DINT(#FS.Intern.ErrorWarning.dwModuleErrorID);
       #SD.ErrorWarning.wError := #FS.ErrorWarning.wError;
       #SD.ErrorWarning.wWarning := #FS.ErrorWarning.wWarning;
       #SD.ErrorWarningReleased := #FS.Intern.ErrorWarningReleased;
   END_REGION

   #SD.iModeActual := #FM.ModeActual;
   #SD.iModuleState := #FS.StateCases.iModule;
   #SD.ProcessValue := #FS.ProcessValues;
   #SD.Recipe := #FS.Recipe;
END_REGION

REGION Network 27 (SCL): Functional Strategy: Mapping to VIS status
   //Module template
   #VIS.CD := #CD;
   #VIS.SD := #SD;
   #VIS.Indicators := #FS.Indicators;
   #VIS.Interlocks := #FM.Interlock;

   //Module specific 
   #VIS.bLimitsSwitchPositiveActivated := #InstanceOEM_LCB_12x_TablePositioning_V2.xHW_LimitSwitchPos;
   #VIS.bLimitsSwitchNegativeActivated := #InstanceOEM_LCB_12x_TablePositioning_V2.xHW_LimitSwitchNeg;
   #VIS.bHomingSensorActivated := #InstanceOEM_LCB_12x_TablePositioning_V2.xHomingSensorActivated;
END_REGION
END_FUNCTION_BLOCK

FUNCTION_BLOCK "CmCommon"   // FB4, SCL
{ S7_Optimized_Access := 'TRUE' }
VERSION : 0.1
   VAR_OUTPUT
      q_stc_sw : "stcCmCommon_SW";
      q_dtlActualPlcSystem_Time : DTL;
      q_rActualPlcCycleTime_Sec : Real;
      q_bSyncBlink : Bool;   // Signal light Indicator blink
      q_bSyncBlinkText : Bool;   // Hmi status text scroll, swap, refresh blink
      q_bSyncPulsText : Bool;   // Text change puls for one cpu cycle
   END_VAR
   VAR_IN_OUT
      iq_Vis : "stcCmCommon_VIS";
   END_VAR
   VAR
      l_bBusyLoadNewTime : Bool;
      ldtl_new_time : DTL;
      lstc_dtl_edit AT ldtl_new_time : Struct
         year : UInt;
         month : USInt;
         day : USInt;
         weekday : USInt;
         hour : USInt;
         minute : USInt;
         second : USInt;
         nanosecond : UDInt;
      END_STRUCT;
      ldtl_prev_time : DTL;   // Need to calculate actual CPU cycle time
      l_InitCpuCycleTimeCalc : Bool;
      l_rTimerSyncBlink_Sec : Real;
      l_bSyncBlink : Bool;
      l_bSyncBlinkText : Bool;
      l_rTimerSyncBlinkText_Sec : Real;
      l_bSyncPulsText : Bool;
      Instance_R_TRIG : R_TRIG;
   END_VAR
   VAR_TEMP
      retval_time_wrt : Int;
      retval_time_act : Int;
      "tt_cycle-time" : Time;
      "ti_cycle-time" : Int;
   END_VAR
BEGIN
   (*****************************************************************************
                           (c) 2018 Maan Engineering b.v.                                    
                                 All rights reserved.                                              

   NAME        :  CmCommon                                             
   FUNCTION    :  Managing the PLC en HMI time and global sync blink en text blink/scroll                                  

   AUTHOR      : Arjan Bovenmars                                 
   DATE        : "Date Created" 2018-11-27
   UPDATE      : See "Last Modified"                                        


   Modification History:                                  By:   Date:    Rev:
   ------------------------------------------------------ --- ---------- ---
   First Version                                         :ABS 2018-11-27 0.0

   *****************************************************************************)//Header
   (***********************************
   Function:  eq_common

   A.Bovenmars
   30-6-2016
   *************************************);
   //Always bit control
   #q_stc_sw.q_bAlwaysFalse  := FALSE;
   #q_stc_sw.q_bAlwaysTrue   := TRUE;

   //Setup system time
   (*Synchrinization OF Time between the PLC cpu AND the HMI exceed over each 60[sec]
   //Synch cycle is a time setting in the global communication of the HMI WinCC program by connection.
   *)
   IF #iq_Vis.stc_NewTimeToSet.iq_bRequestLoadNewTime AND NOT #l_bBusyLoadNewTime THEN
       #iq_Vis.stc_NewTimeToSet.iq_bRequestLoadNewTime := false; //clear the aceppted request.
       #l_bBusyLoadNewTime := true; // set the memory that request is set. 
       #lstc_dtl_edit.year := #iq_Vis.stc_NewTimeToSet.year;
       #lstc_dtl_edit.month := #iq_Vis.stc_NewTimeToSet.month;
       #lstc_dtl_edit.weekday := #iq_Vis.stc_NewTimeToSet.weekday;
       #lstc_dtl_edit.day := #iq_Vis.stc_NewTimeToSet.day;
       #lstc_dtl_edit.hour := #iq_Vis.stc_NewTimeToSet.hour;
       #lstc_dtl_edit.minute := #iq_Vis.stc_NewTimeToSet.minute;

   ELSIF #l_bBusyLoadNewTime AND NOT #iq_Vis.stc_NewTimeToSet.iq_bRequestLoadNewTime THEN
       #retval_time_wrt := WR_SYS_T(#ldtl_new_time);
       #l_bBusyLoadNewTime := false;
   END_IF;//Set new system time

   //Read sytem PLC time and write to PLC output and visualisation
   #retval_time_act := RD_SYS_T(#q_dtlActualPlcSystem_Time);   
   #iq_Vis.q_dtlActualPlcSystemTime := #q_dtlActualPlcSystem_Time;

   //CPU cyle time calculation
   IF NOT #l_InitCpuCycleTimeCalc THEN
       #ldtl_prev_time := #q_dtlActualPlcSystem_Time;
       #l_InitCpuCycleTimeCalc := TRUE;
   END_IF;

   #"tt_cycle-time" := T_DIFF(IN1 := #q_dtlActualPlcSystem_Time, IN2 := #ldtl_prev_time); //Difference between previous and new DTL time
   #ldtl_prev_time := #q_dtlActualPlcSystem_Time; //Set the current time as previous time for the next cpu cycle.
   #"ti_cycle-time" := TIME_TO_INT(#"tt_cycle-time");//Set the time into a integer
   #q_rActualPlcCycleTime_Sec := ((INT_TO_REAL(#"ti_cycle-time")) / 1000);// set the time into seconds in a real format and put as global output
   #iq_Vis.q_rActualPlcCycleTime_Sec := #q_rActualPlcCycleTime_Sec;
   //-------------------------------------------------------------
   //

   //Synchronization blink for indicator for the compleet unit or process-cell
   IF #l_rTimerSyncBlink_Sec >= 0.5 THEN
       #l_rTimerSyncBlink_Sec := 0;//clear timer
       #l_bSyncBlink := NOT #l_bSyncBlink;
   ELSE
       #l_rTimerSyncBlink_Sec := #l_rTimerSyncBlink_Sec + #q_rActualPlcCycleTime_Sec;
   END_IF;
   #q_bSyncBlink := #l_bSyncBlink; //copy local to global

   //Synchronization HMi text blink 
   IF #l_rTimerSyncBlinkText_Sec >= 1.8 THEN
       #l_rTimerSyncBlinkText_Sec := 0;
       #l_bSyncBlinkText := NOT #l_bSyncBlinkText;
   ELSE
       #l_rTimerSyncBlinkText_Sec := #l_rTimerSyncBlinkText_Sec + #q_rActualPlcCycleTime_Sec;
   END_IF;
   #q_bSyncBlinkText := #l_bSyncBlinkText;

   //Synchronization HMi text blink puls
   #Instance_R_TRIG(CLK:=#l_bSyncBlinkText,
                    Q=>#l_bSyncPulsText);
   #q_bSyncPulsText := #l_bSyncPulsText;



   //Write to global StatusWord
   #q_stc_sw.q_bSyncBlink := #q_bSyncBlink;
   #q_stc_sw.q_bSyncBlinkText := #q_bSyncBlinkText;
   #q_stc_sw.q_dtlActualPlcSystem_Time := #q_dtlActualPlcSystem_Time;
   #q_stc_sw.q_rActualPlcCycleTime_Sec := #q_rActualPlcCycleTime_Sec;
   #q_stc_sw.q_bSyncPulsText := #q_bSyncPulsText;
END_FUNCTION_BLOCK

ORGANIZATION_BLOCK "Main"   // OB1, FBD, ProgramCycle
TITLE = "Main Program Sweep (Cycle)"
{ S7_Optimized_Access := 'TRUE' }
VERSION : 0.1
   VAR_INPUT
      Initial_Call : Bool;   // Initial call of this OB
      Remanence : Bool;   // =True, if remanent data are available
   END_VAR
BEGIN

REGION Network 1: CmCommon
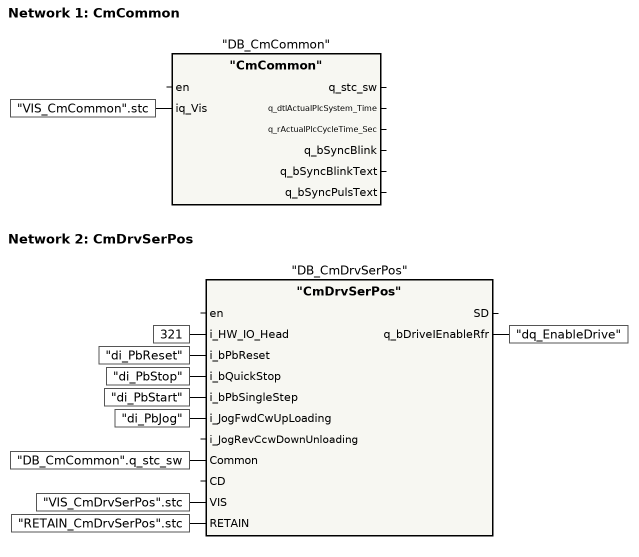
   "DB_CmCommon"(iq_Vis := "VIS_CmCommon".stc);   // "CmCommon"
END_REGION

REGION Network 2: CmDrvSerPos
   "DB_CmDrvSerPos"(i_HW_IO_Head := 321,   // "CmDrvSerPos"
                    i_bPbReset := "di_PbReset",
                    i_bQuickStop := "di_PbStop",
                    i_bPbSingleStep := "di_PbStart",
                    i_JogFwdCwUpLoading := "di_PbJog",
                    Common := "DB_CmCommon".q_stc_sw,
                    VIS := "VIS_CmDrvSerPos".stc,
                    RETAIN := "RETAIN_CmDrvSerPos".stc,
                    q_bDriveIEnableRfr => "dq_EnableDrive");
END_REGION
END_ORGANIZATION_BLOCK

// folder: OEM

